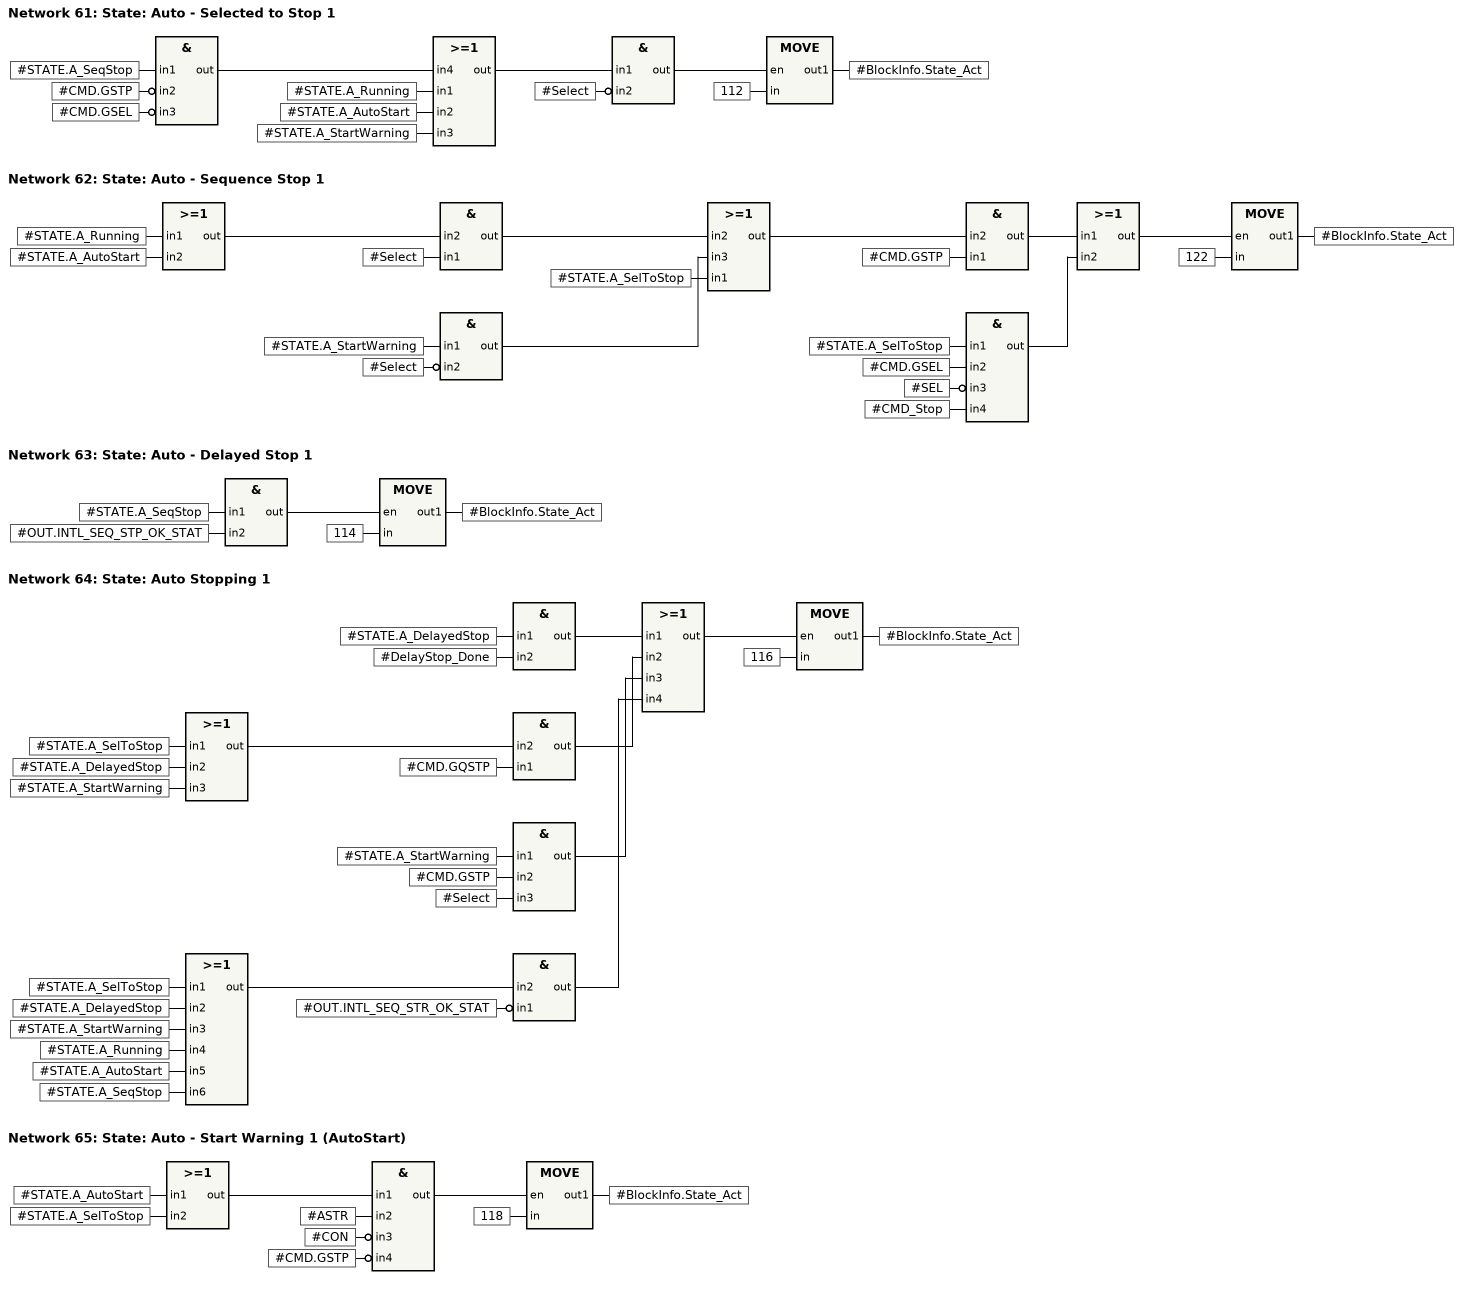
   IF ((#STATE.A_SeqStop AND NOT #CMD.GSTP AND NOT #CMD.GSEL) OR #STATE.A_Running OR #STATE.A_AutoStart OR #STATE.A_StartWarning) AND NOT #Select THEN
       #BlockInfo.State_Act := 112;
   END_IF;
END_REGION

REGION Network 62: State: Auto - Sequence Stop 1
   IF ((((#STATE.A_Running OR #STATE.A_AutoStart) AND #Select) OR (#STATE.A_StartWarning AND NOT #Select) OR #STATE.A_SelToStop) AND #CMD.GSTP) OR (#STATE.A_SelToStop AND #CMD.GSEL AND NOT #SEL AND #CMD_Stop) THEN
       #BlockInfo.State_Act := 122;
   END_IF;
END_REGION

REGION Network 63: State: Auto - Delayed Stop 1
   IF #STATE.A_SeqStop AND #OUT.INTL_SEQ_STP_OK_STAT THEN #BlockInfo.State_Act := 114; END_IF;
END_REGION

REGION Network 64: State: Auto Stopping 1
   IF (#STATE.A_DelayedStop AND #DelayStop_Done) OR ((#STATE.A_SelToStop OR #STATE.A_DelayedStop OR #STATE.A_StartWarning) AND #CMD.GQSTP) OR (#STATE.A_StartWarning AND #CMD.GSTP AND #Select) OR ((#STATE.A_SelToStop OR #STATE.A_DelayedStop OR #STATE.A_StartWarning OR #STATE.A_Running OR #STATE.A_AutoStart OR #STATE.A_SeqStop) AND NOT #OUT.INTL_SEQ_STR_OK_STAT) THEN
       #BlockInfo.State_Act := 116;
   END_IF;
END_REGION

REGION Network 65: State: Auto - Start Warning 1 (AutoStart)
   IF (#STATE.A_AutoStart OR #STATE.A_SelToStop) AND #ASTR AND NOT #CON AND NOT #CMD.GSTP THEN
       #BlockInfo.State_Act := 118;
   END_IF;
END_REGION

REGION Network 66
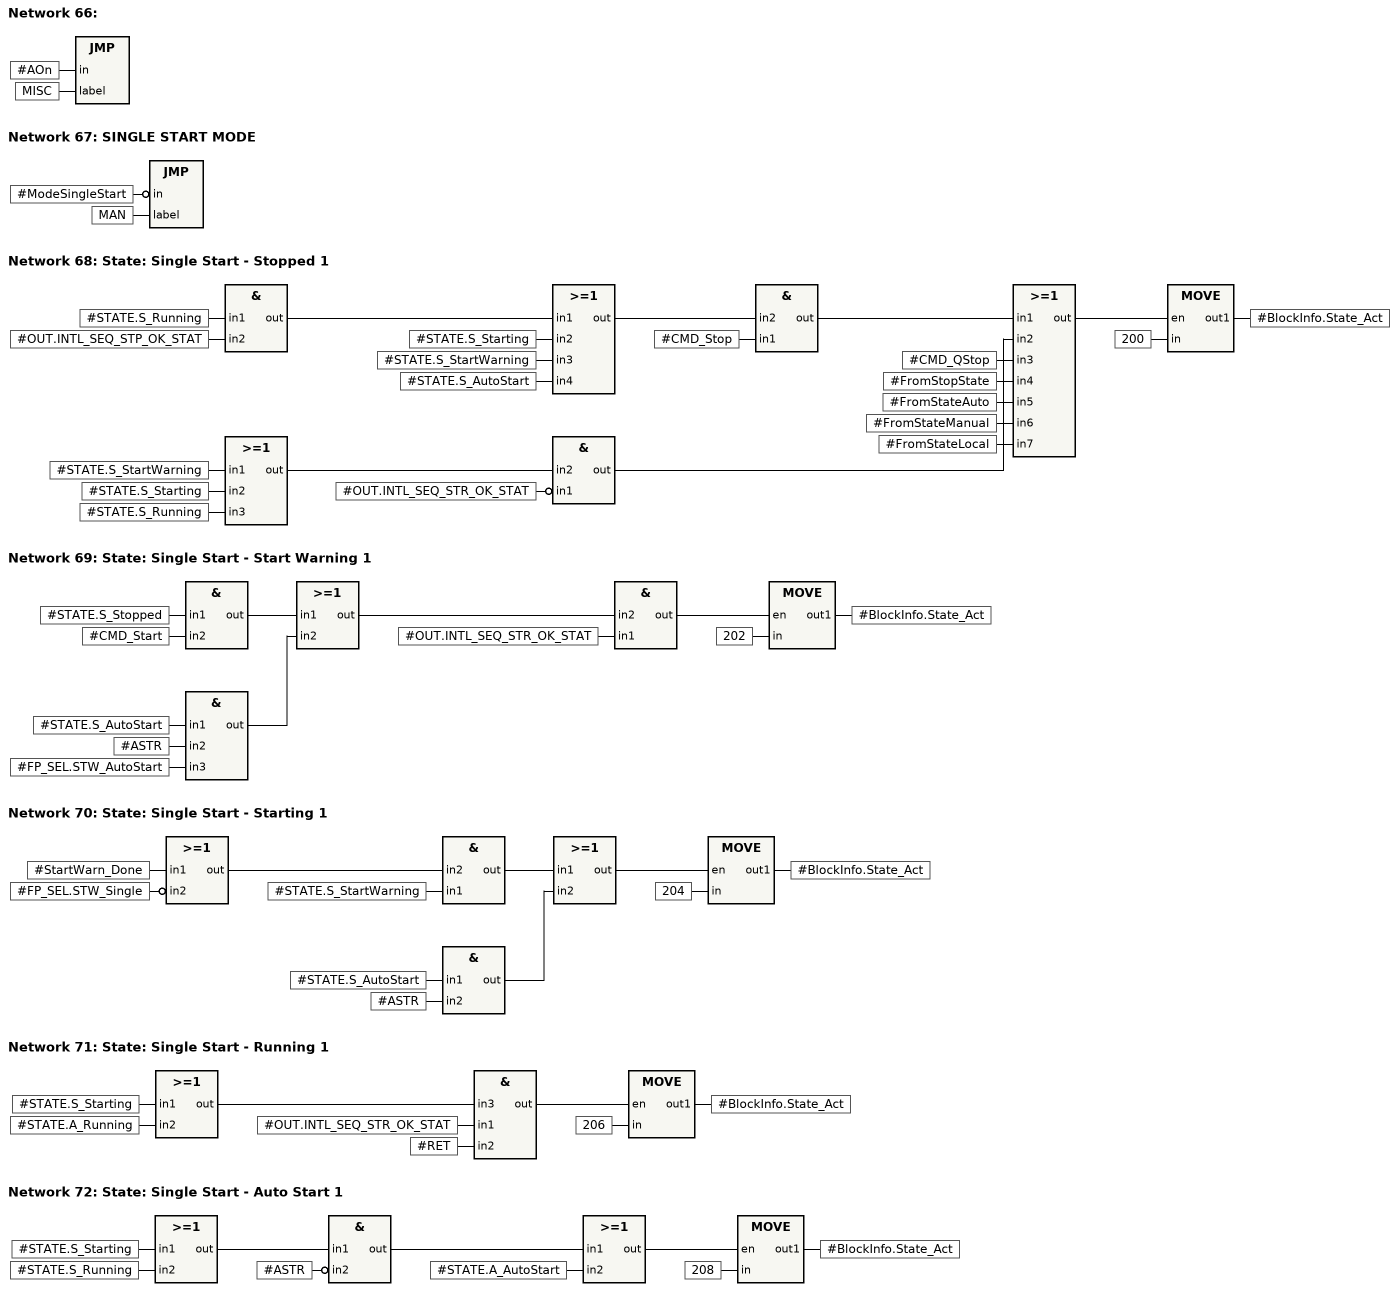
   IF #AOn THEN GOTO MISC; END_IF;
END_REGION

REGION Network 67: SINGLE START MODE
   SS1:
   IF NOT #ModeSingleStart THEN GOTO MAN; END_IF;
END_REGION

REGION Network 68: State: Single Start - Stopped 1
   IF (((#STATE.S_Running AND #OUT.INTL_SEQ_STP_OK_STAT) OR #STATE.S_Starting OR #STATE.S_StartWarning OR #STATE.S_AutoStart) AND #CMD_Stop) OR ((#STATE.S_StartWarning OR #STATE.S_Starting OR #STATE.S_Running) AND NOT #OUT.INTL_SEQ_STR_OK_STAT) OR #CMD_QStop OR #FromStopState OR #FromStateAuto OR #FromStateManual OR #FromStateLocal THEN
       #BlockInfo.State_Act := 200;
   END_IF;
END_REGION

REGION Network 69: State: Single Start - Start Warning 1
   IF ((#STATE.S_Stopped AND #CMD_Start) OR (#STATE.S_AutoStart AND #ASTR AND #FP_SEL.STW_AutoStart)) AND #OUT.INTL_SEQ_STR_OK_STAT THEN
       #BlockInfo.State_Act := 202;
   END_IF;
END_REGION

REGION Network 70: State: Single Start - Starting 1
   IF ((#StartWarn_Done OR NOT #FP_SEL.STW_Single) AND #STATE.S_StartWarning) OR (#STATE.S_AutoStart AND #ASTR) THEN
       #BlockInfo.State_Act := 204;
   END_IF;
END_REGION

REGION Network 71: State: Single Start - Running 1
   IF (#STATE.S_Starting OR #STATE.A_Running) AND #OUT.INTL_SEQ_STR_OK_STAT AND #RET THEN
       #BlockInfo.State_Act := 206;
   END_IF;
END_REGION

REGION Network 72: State: Single Start - Auto Start 1
   IF ((#STATE.S_Starting OR #STATE.S_Running) AND NOT #ASTR) OR #STATE.A_AutoStart THEN
       #BlockInfo.State_Act := 208;
   END_IF;
END_REGION

REGION Network 73
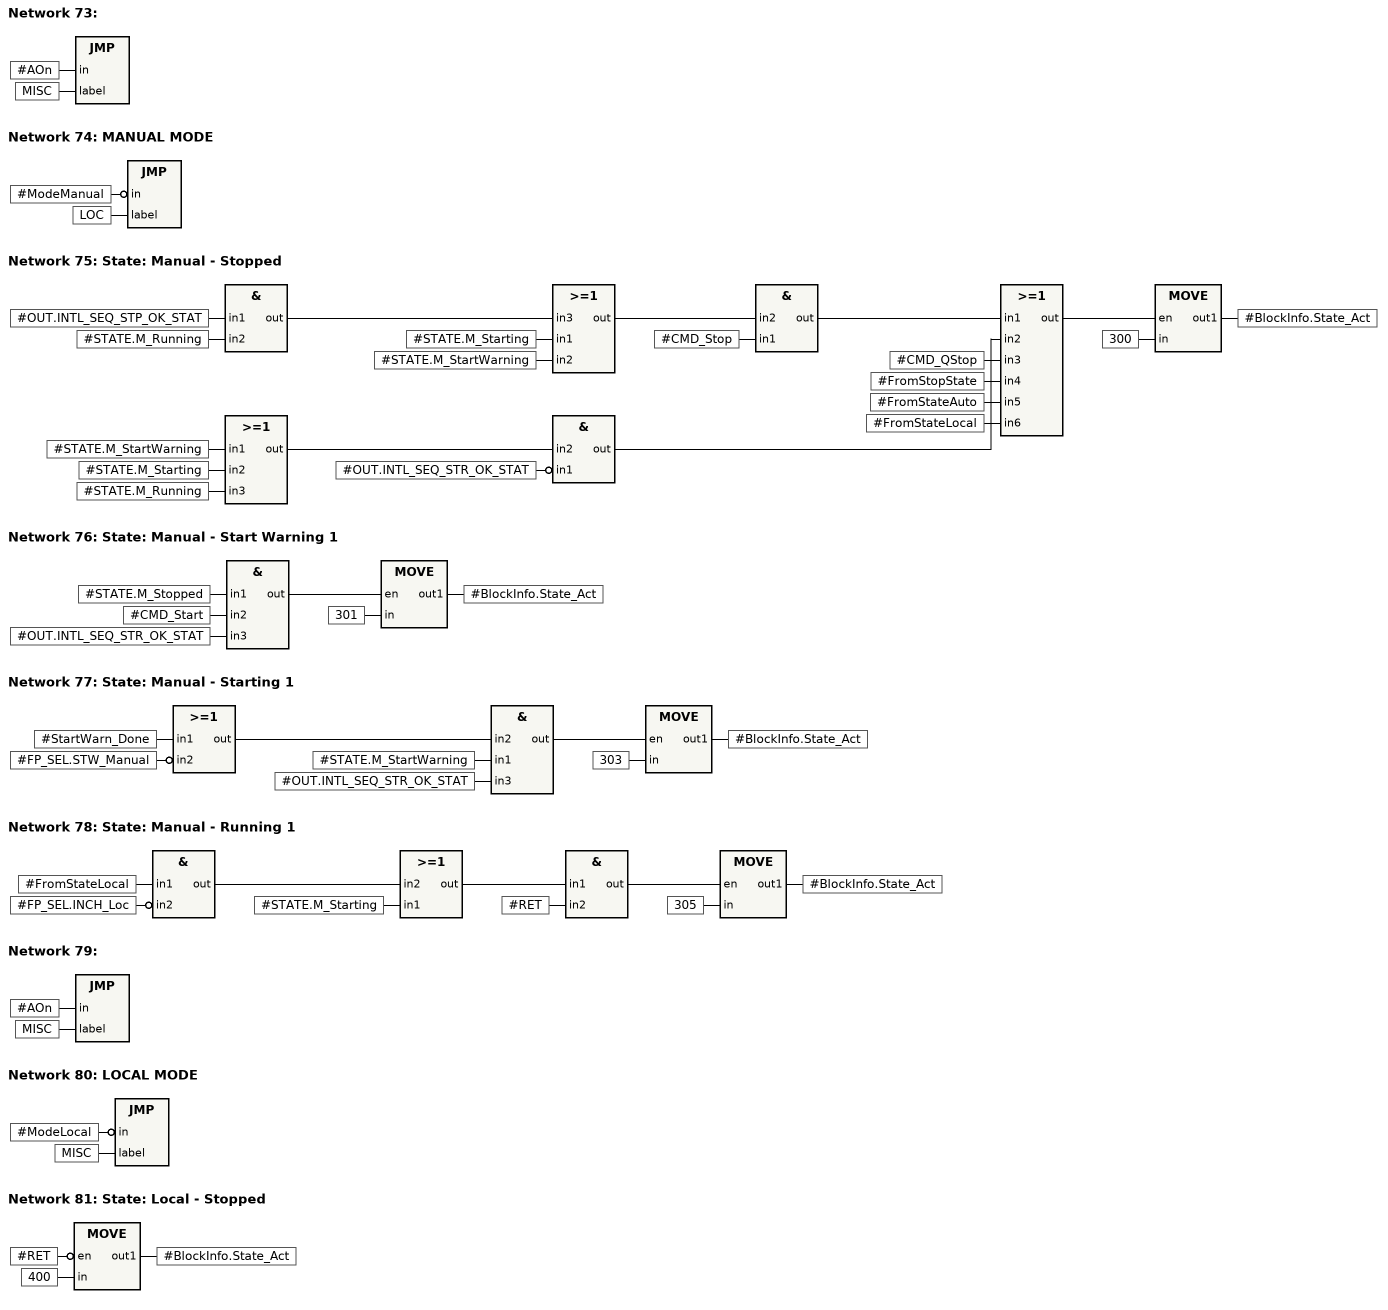
   IF #AOn THEN GOTO MISC; END_IF;
END_REGION

REGION Network 74: MANUAL MODE
   MAN:
   IF NOT #ModeManual THEN GOTO LOC; END_IF;
END_REGION

REGION Network 75: State: Manual - Stopped
   IF (((#OUT.INTL_SEQ_STP_OK_STAT AND #STATE.M_Running) OR #STATE.M_Starting OR #STATE.M_StartWarning) AND #CMD_Stop) OR ((#STATE.M_StartWarning OR #STATE.M_Starting OR #STATE.M_Running) AND NOT #OUT.INTL_SEQ_STR_OK_STAT) OR #CMD_QStop OR #FromStopState OR #FromStateAuto OR #FromStateLocal THEN
       #BlockInfo.State_Act := 300;
   END_IF;
END_REGION

REGION Network 76: State: Manual - Start Warning 1
   IF #STATE.M_Stopped AND #CMD_Start AND #OUT.INTL_SEQ_STR_OK_STAT THEN #BlockInfo.State_Act := 301; END_IF;
END_REGION

REGION Network 77: State: Manual - Starting 1
   IF (#StartWarn_Done OR NOT #FP_SEL.STW_Manual) AND #STATE.M_StartWarning AND #OUT.INTL_SEQ_STR_OK_STAT THEN
       #BlockInfo.State_Act := 303;
   END_IF;
END_REGION

REGION Network 78: State: Manual - Running 1
   IF ((#FromStateLocal AND NOT #FP_SEL.INCH_Loc) OR #STATE.M_Starting) AND #RET THEN
       #BlockInfo.State_Act := 305;
   END_IF;
END_REGION

REGION Network 79
   IF #AOn THEN GOTO MISC; END_IF;
END_REGION

REGION Network 80: LOCAL MODE
   LOC:
   IF NOT #ModeLocal THEN GOTO MISC; END_IF;
END_REGION

REGION Network 81: State: Local - Stopped
   IF NOT #RET THEN #BlockInfo.State_Act := 400; END_IF;
END_REGION

REGION Network 82: State: Local Running 1
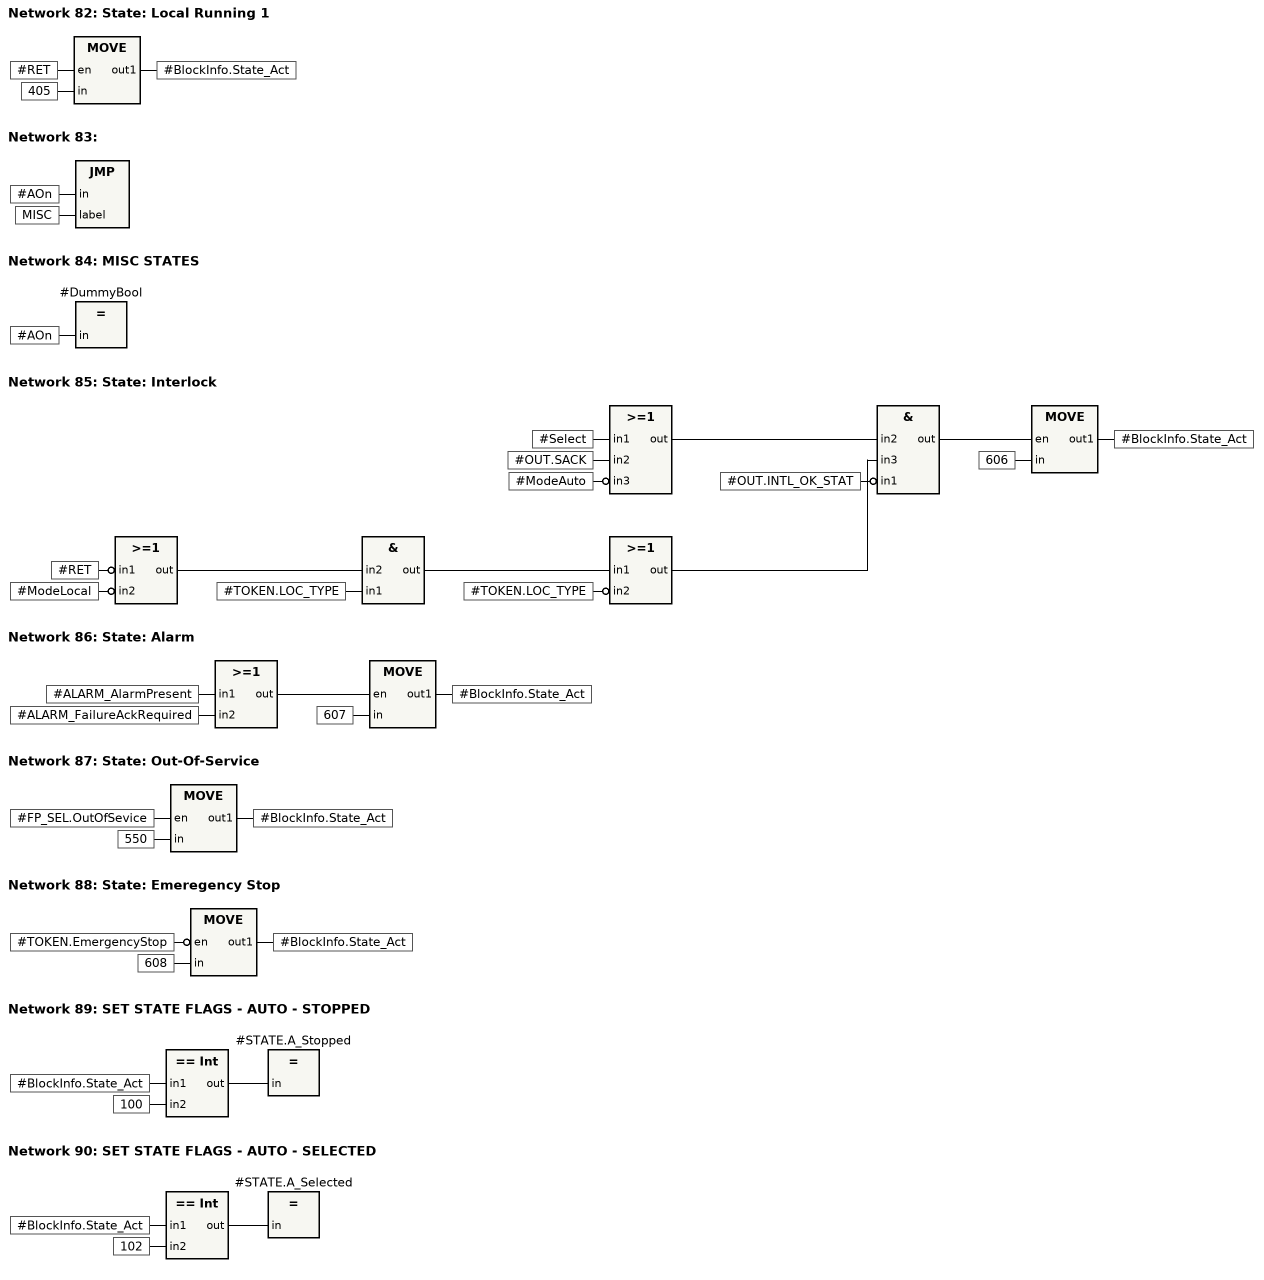
   IF #RET THEN #BlockInfo.State_Act := 405; END_IF;
END_REGION

REGION Network 83
   IF #AOn THEN GOTO MISC; END_IF;
END_REGION

REGION Network 84: MISC STATES
   MISC:
   #DummyBool := #AOn;
END_REGION

REGION Network 85: State: Interlock
   IF (#Select OR #OUT.SACK OR NOT #ModeAuto) AND (((NOT #RET OR NOT #ModeLocal) AND #TOKEN.LOC_TYPE) OR NOT #TOKEN.LOC_TYPE) AND NOT #OUT.INTL_OK_STAT THEN
       #BlockInfo.State_Act := 606;
   END_IF;
END_REGION

REGION Network 86: State: Alarm
   IF #ALARM_AlarmPresent OR #ALARM_FailureAckRequired THEN #BlockInfo.State_Act := 607; END_IF;
END_REGION

REGION Network 87: State: Out-Of-Service
   IF #FP_SEL.OutOfSevice THEN #BlockInfo.State_Act := 550; END_IF;
END_REGION

REGION Network 88: State: Emeregency Stop
   IF NOT #TOKEN.EmergencyStop THEN #BlockInfo.State_Act := 608; END_IF;
END_REGION

REGION Network 89: SET STATE FLAGS - AUTO - STOPPED
   #STATE.A_Stopped := #BlockInfo.State_Act = 100;
END_REGION

REGION Network 90: SET STATE FLAGS - AUTO - SELECTED
   #STATE.A_Selected := #BlockInfo.State_Act = 102;
END_REGION

REGION Network 91: SET STATE FLAGS - AUTO - SEQ START
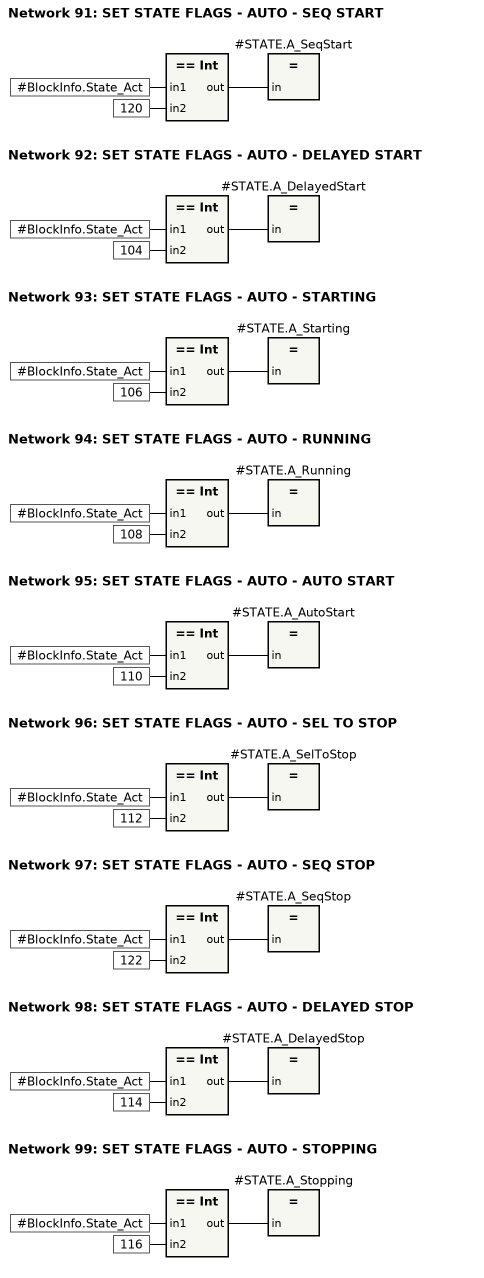
   #STATE.A_SeqStart := #BlockInfo.State_Act = 120;
END_REGION

REGION Network 92: SET STATE FLAGS - AUTO - DELAYED START
   #STATE.A_DelayedStart := #BlockInfo.State_Act = 104;
END_REGION

REGION Network 93: SET STATE FLAGS - AUTO - STARTING
   #STATE.A_Starting := #BlockInfo.State_Act = 106;
END_REGION

REGION Network 94: SET STATE FLAGS - AUTO - RUNNING
   #STATE.A_Running := #BlockInfo.State_Act = 108;
END_REGION

REGION Network 95: SET STATE FLAGS - AUTO - AUTO START
   #STATE.A_AutoStart := #BlockInfo.State_Act = 110;
END_REGION

REGION Network 96: SET STATE FLAGS - AUTO - SEL TO STOP
   #STATE.A_SelToStop := #BlockInfo.State_Act = 112;
END_REGION

REGION Network 97: SET STATE FLAGS - AUTO - SEQ STOP
   #STATE.A_SeqStop := #BlockInfo.State_Act = 122;
END_REGION

REGION Network 98: SET STATE FLAGS - AUTO - DELAYED STOP
   #STATE.A_DelayedStop := #BlockInfo.State_Act = 114;
END_REGION

REGION Network 99: SET STATE FLAGS - AUTO - STOPPING
   #STATE.A_Stopping := #BlockInfo.State_Act = 116;
END_REGION

REGION Network 100: SET STATE FLAGS - AUTO - START WARNING
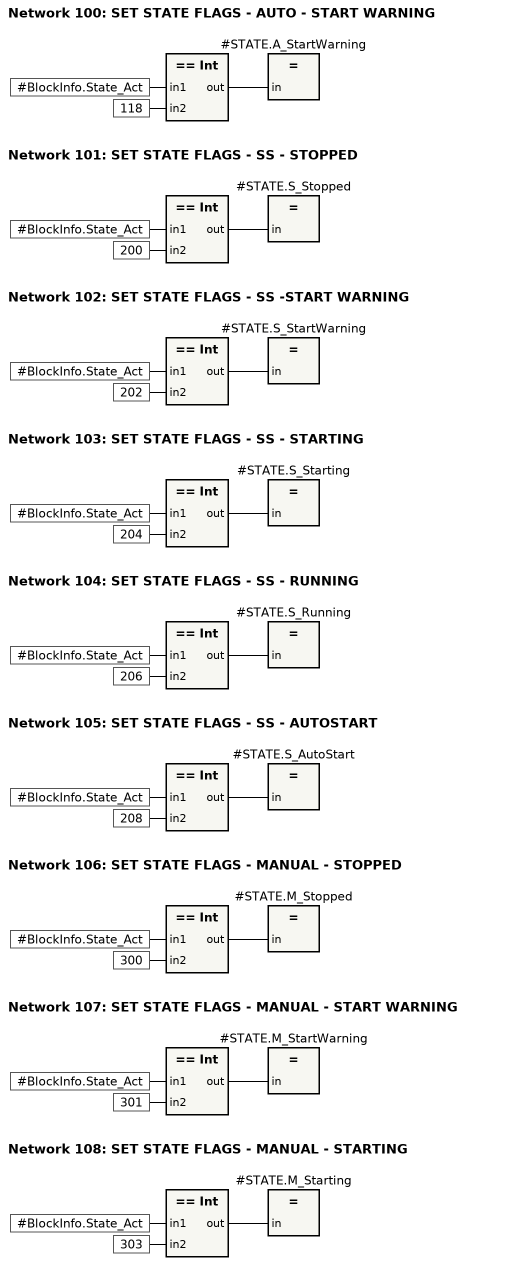
   #STATE.A_StartWarning := #BlockInfo.State_Act = 118;
END_REGION

REGION Network 101: SET STATE FLAGS - SS - STOPPED
   #STATE.S_Stopped := #BlockInfo.State_Act = 200;
END_REGION

REGION Network 102: SET STATE FLAGS - SS -START WARNING
   #STATE.S_StartWarning := #BlockInfo.State_Act = 202;
END_REGION

REGION Network 103: SET STATE FLAGS - SS - STARTING
   #STATE.S_Starting := #BlockInfo.State_Act = 204;
END_REGION

REGION Network 104: SET STATE FLAGS - SS - RUNNING
   #STATE.S_Running := #BlockInfo.State_Act = 206;
END_REGION

REGION Network 105: SET STATE FLAGS - SS - AUTOSTART
   #STATE.S_AutoStart := #BlockInfo.State_Act = 208;
END_REGION

REGION Network 106: SET STATE FLAGS - MANUAL - STOPPED
   #STATE.M_Stopped := #BlockInfo.State_Act = 300;
END_REGION

REGION Network 107: SET STATE FLAGS - MANUAL - START WARNING
   #STATE.M_StartWarning := #BlockInfo.State_Act = 301;
END_REGION

REGION Network 108: SET STATE FLAGS - MANUAL - STARTING
   #STATE.M_Starting := #BlockInfo.State_Act = 303;
END_REGION

REGION Network 109: SET STATE FLAGS - MANUAL - RUNNING
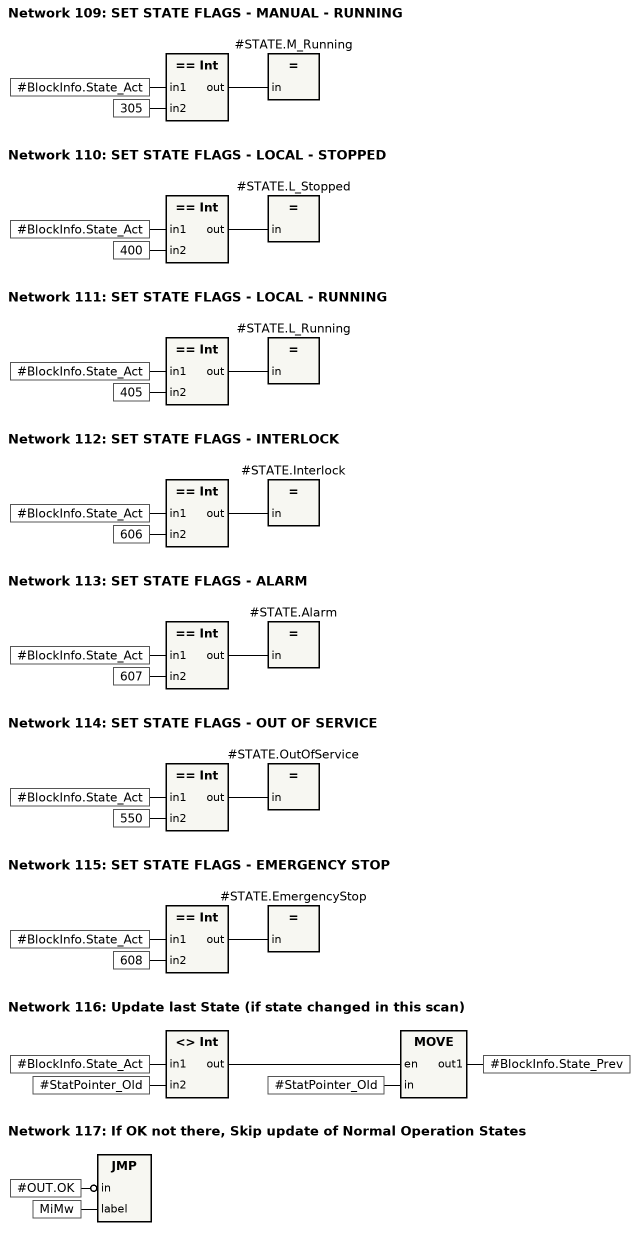
   #STATE.M_Running := #BlockInfo.State_Act = 305;
END_REGION

REGION Network 110: SET STATE FLAGS - LOCAL - STOPPED
   #STATE.L_Stopped := #BlockInfo.State_Act = 400;
END_REGION

REGION Network 111: SET STATE FLAGS - LOCAL - RUNNING
   #STATE.L_Running := #BlockInfo.State_Act = 405;
END_REGION

REGION Network 112: SET STATE FLAGS - INTERLOCK
   #STATE.Interlock := #BlockInfo.State_Act = 606;
END_REGION

REGION Network 113: SET STATE FLAGS - ALARM
   #STATE.Alarm := #BlockInfo.State_Act = 607;
END_REGION

REGION Network 114: SET STATE FLAGS - OUT OF SERVICE
   #STATE.OutOfService := #BlockInfo.State_Act = 550;
END_REGION

REGION Network 115: SET STATE FLAGS - EMERGENCY STOP
   #STATE.EmergencyStop := #BlockInfo.State_Act = 608;
END_REGION

REGION Network 116: Update last State (if state changed in this scan)
   IF #BlockInfo.State_Act <> #StatPointer_Old THEN #BlockInfo.State_Prev := #StatPointer_Old; END_IF;
END_REGION

REGION Network 117: If OK not there, Skip update of Normal Operation States
   // Build 006 - 30.09.2020 (EXTBOB): Skipped Normal MSW status update in case of Alarm Condition, Newly Added
   IF NOT #OUT.OK THEN GOTO MiMw; END_IF;
END_REGION

REGION Network 118: UPDATE MSW
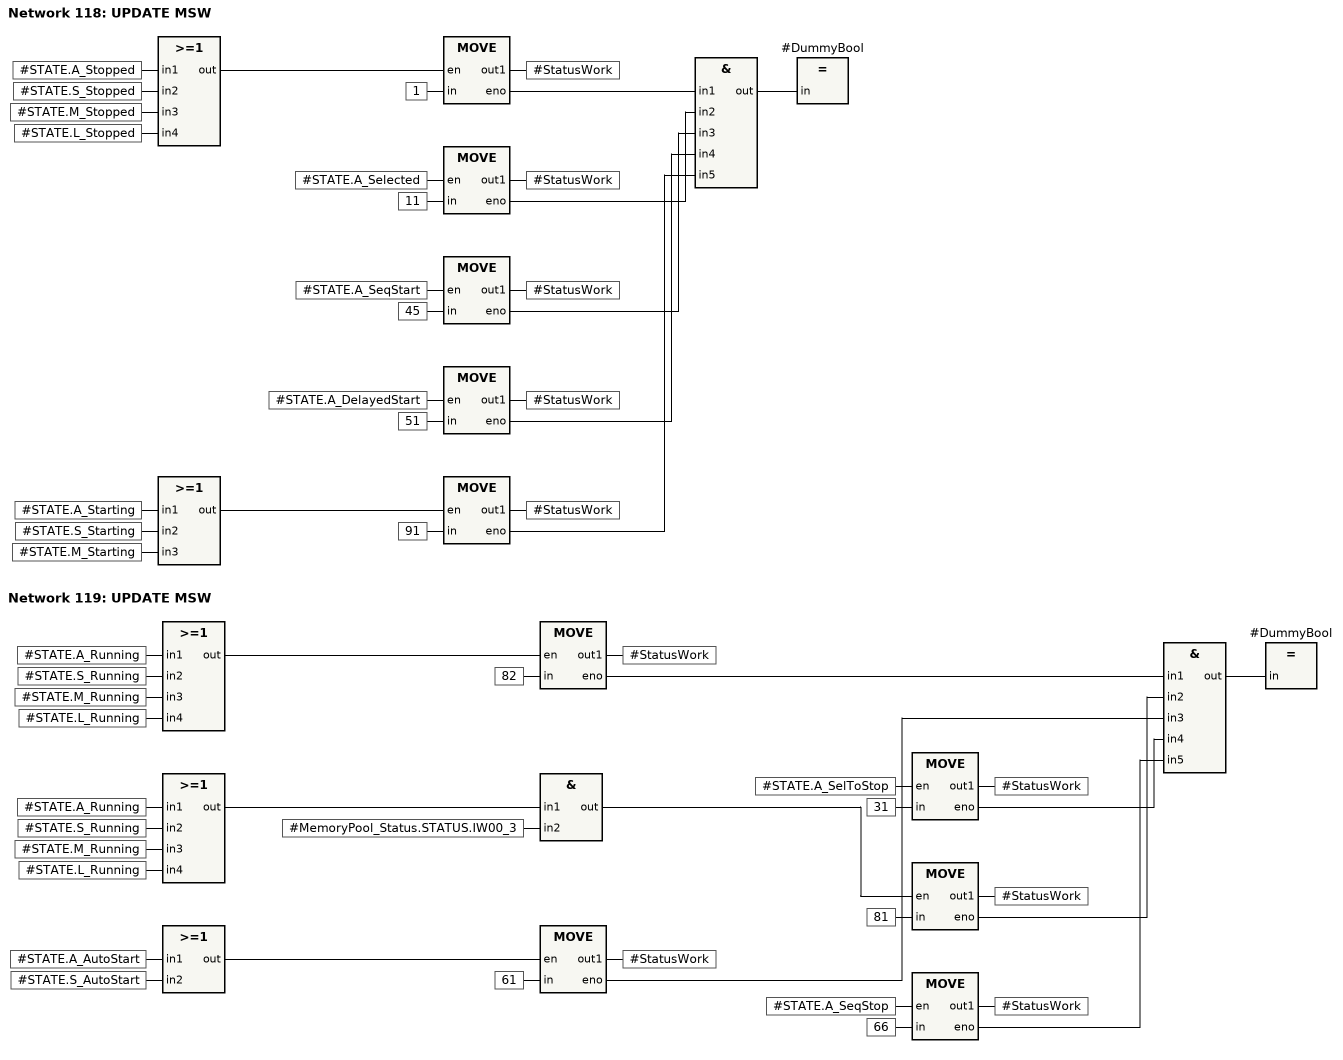
   // ENO of a box is taken as its EN; it also drops when the box reports an error
   #_w1 := #STATE.A_Stopped OR #STATE.S_Stopped OR #STATE.M_Stopped OR #STATE.L_Stopped;
   IF #_w1 THEN #StatusWork := 1; END_IF;
   IF #STATE.A_Selected THEN #StatusWork := 11; END_IF;
   IF #STATE.A_SeqStart THEN #StatusWork := 45; END_IF;
   IF #STATE.A_DelayedStart THEN #StatusWork := 51; END_IF;
   #_w2 := #STATE.A_Starting OR #STATE.S_Starting OR #STATE.M_Starting;
   IF #_w2 THEN #StatusWork := 91; END_IF;
   #DummyBool := #_w1 AND #STATE.A_Selected AND #STATE.A_SeqStart AND #STATE.A_DelayedStart AND #_w2;
END_REGION

REGION Network 119: UPDATE MSW
   // ENO of a box is taken as its EN; it also drops when the box reports an error
   #_w1 := #STATE.A_Running OR #STATE.S_Running OR #STATE.M_Running OR #STATE.L_Running;
   IF #_w1 THEN #StatusWork := 82; END_IF;
   #_w2 := (#STATE.A_Running OR #STATE.S_Running OR #STATE.M_Running OR #STATE.L_Running) AND #MemoryPool_Status.STATUS.IW00_3;
   IF #_w2 THEN #StatusWork := 81; END_IF;
   #_w3 := #STATE.A_AutoStart OR #STATE.S_AutoStart;
   IF #_w3 THEN #StatusWork := 61; END_IF;
   IF #STATE.A_SelToStop THEN #StatusWork := 31; END_IF;
   IF #STATE.A_SeqStop THEN #StatusWork := 66; END_IF;
   #DummyBool := #_w1 AND #_w2 AND #_w3 AND #STATE.A_SelToStop AND #STATE.A_SeqStop;
END_REGION

REGION Network 120
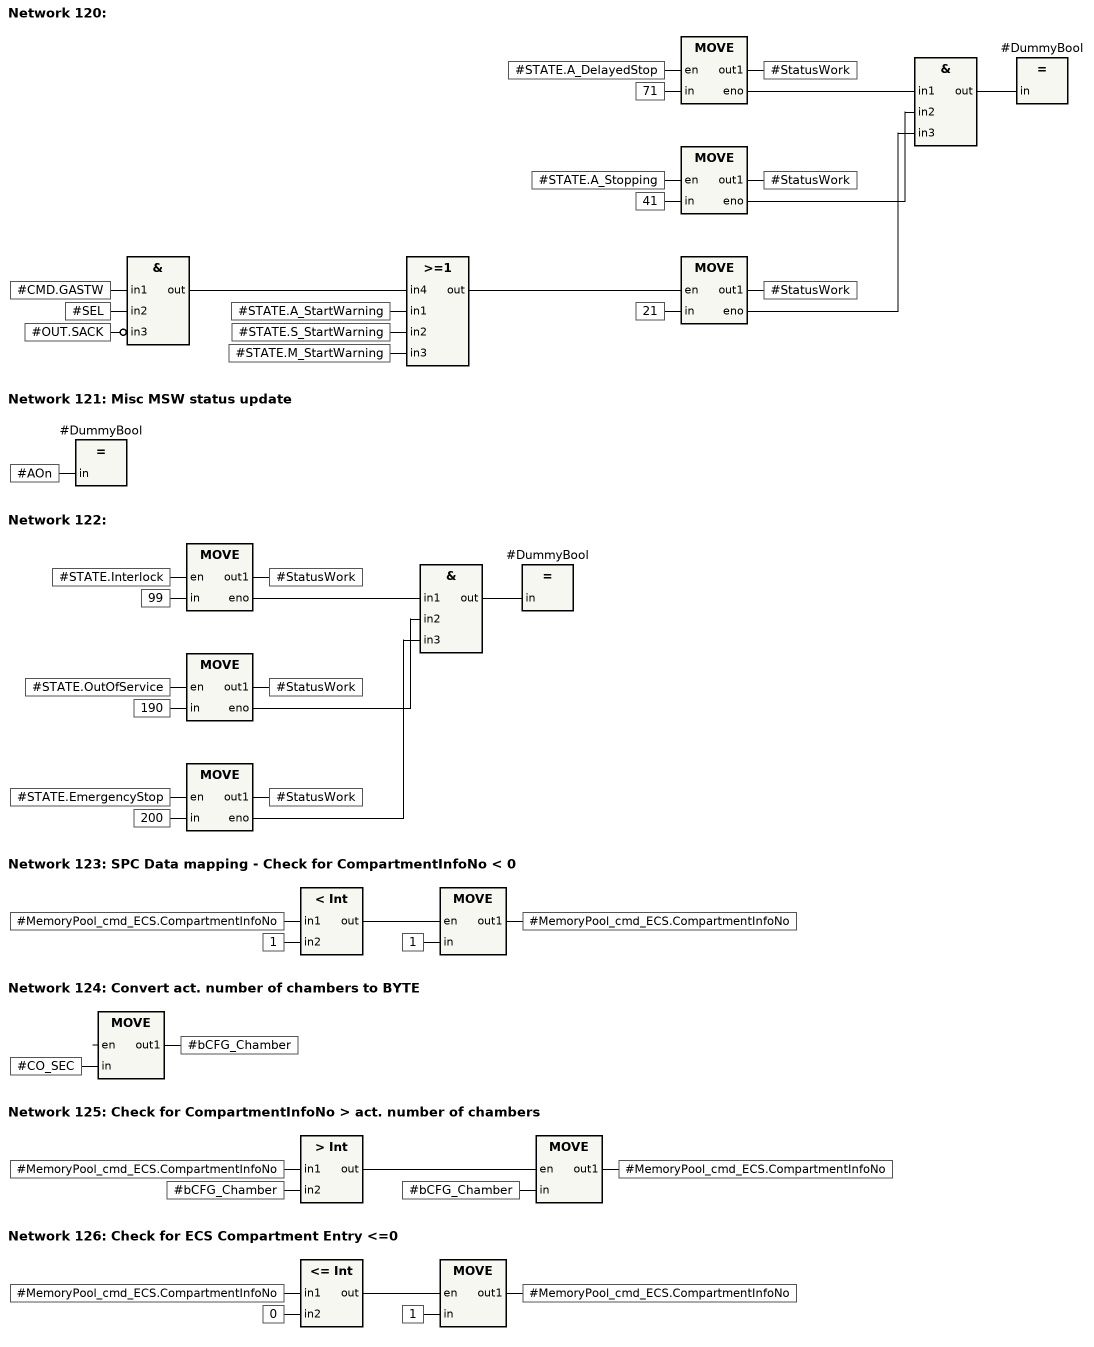
   // ENO of a box is taken as its EN; it also drops when the box reports an error
   IF #STATE.A_DelayedStop THEN #StatusWork := 71; END_IF;
   IF #STATE.A_Stopping THEN #StatusWork := 41; END_IF;
   #_w1 := (#CMD.GASTW AND #SEL AND NOT #OUT.SACK) OR #STATE.A_StartWarning OR #STATE.S_StartWarning OR #STATE.M_StartWarning;
   IF #_w1 THEN #StatusWork := 21; END_IF;
   #DummyBool := #STATE.A_DelayedStop AND #STATE.A_Stopping AND #_w1;
END_REGION

REGION Network 121: Misc MSW status update
   // Build 006 - 30.09.2020 (EXTBOB): Skipped Normal MSW status update in case of Alarm Condition, Newly Added
   MiMw:
   #DummyBool := #AOn;
END_REGION

REGION Network 122
   // ENO of a box is taken as its EN; it also drops when the box reports an error
   IF #STATE.Interlock THEN #StatusWork := 99; END_IF;
   IF #STATE.OutOfService THEN #StatusWork := 190; END_IF;
   IF #STATE.EmergencyStop THEN #StatusWork := 200; END_IF;
   #DummyBool := #STATE.Interlock AND #STATE.OutOfService AND #STATE.EmergencyStop;
END_REGION

REGION Network 123: SPC Data mapping - Check for CompartmentInfoNo < 0
   IF #MemoryPool_cmd_ECS.CompartmentInfoNo < 1 THEN #MemoryPool_cmd_ECS.CompartmentInfoNo := 1; END_IF;
END_REGION

REGION Network 124: Convert act. number of chambers to BYTE
   #bCFG_Chamber := #CO_SEC;
END_REGION

REGION Network 125: Check for CompartmentInfoNo > act. number of chambers
   IF #MemoryPool_cmd_ECS.CompartmentInfoNo > #bCFG_Chamber THEN
       #MemoryPool_cmd_ECS.CompartmentInfoNo := #bCFG_Chamber;
   END_IF;
END_REGION

REGION Network 126: Check for ECS Compartment Entry <=0
   IF #MemoryPool_cmd_ECS.CompartmentInfoNo <= 0 THEN #MemoryPool_cmd_ECS.CompartmentInfoNo := 1; END_IF;
END_REGION

REGION Network 127: Convert IO_Addr from INT to WORD
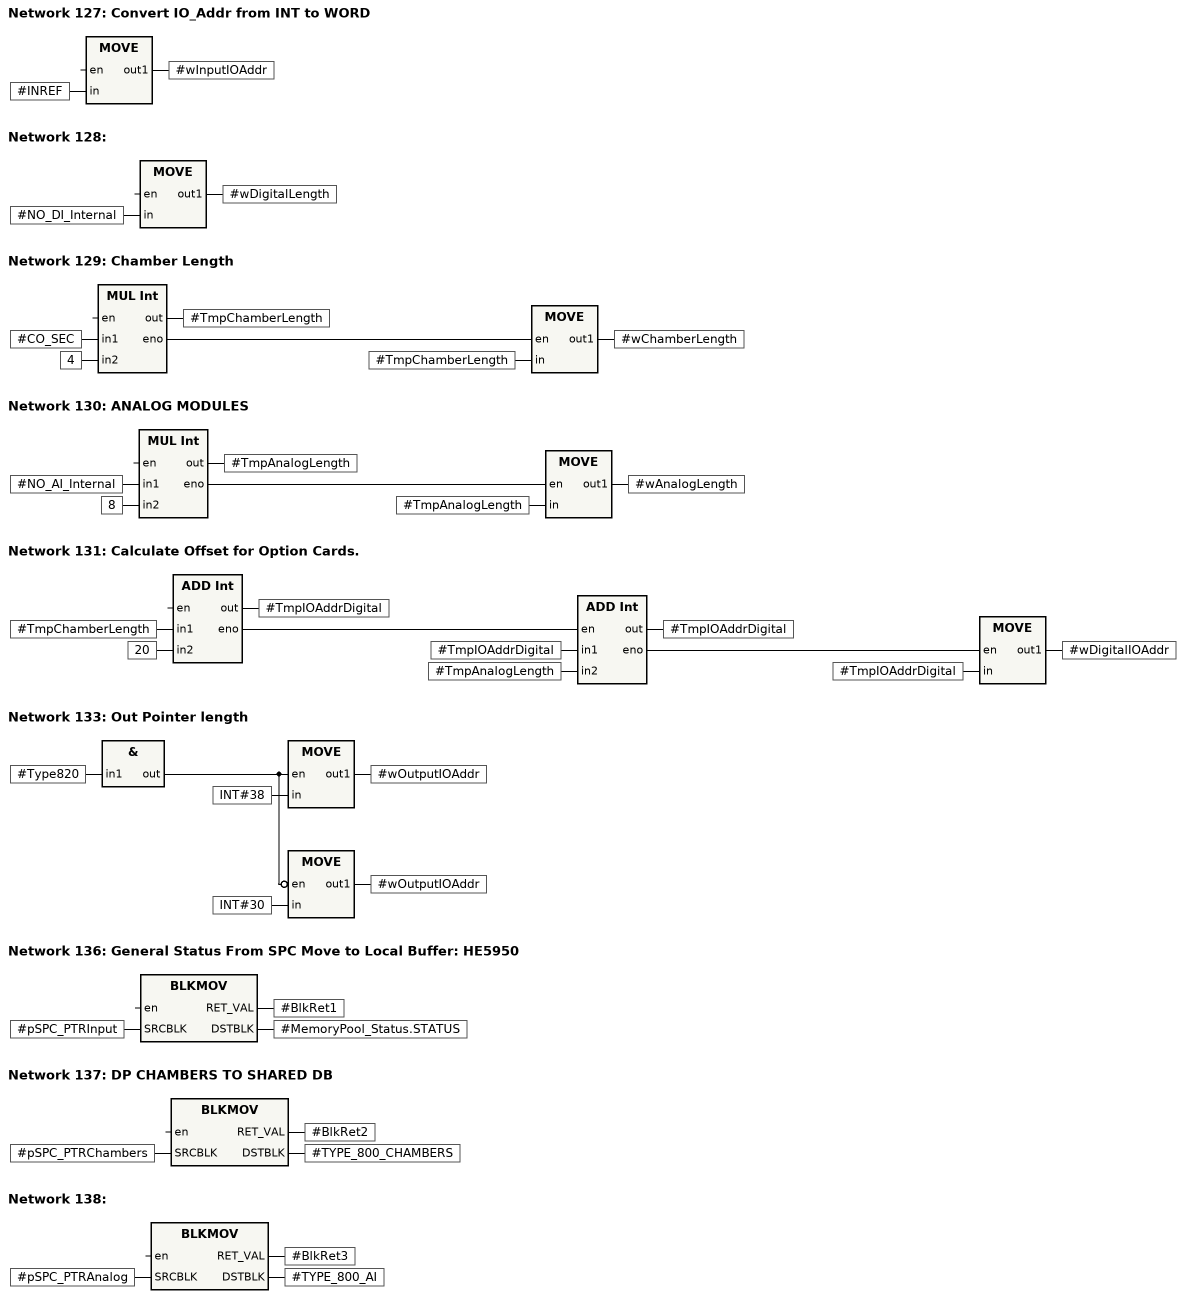
   #wInputIOAddr := #INREF;
END_REGION

REGION Network 128
   // Build 007 - 03.12.2020 (VIV-IN): NO_AI_Internal changed to NO_DI_Internal typo 
   // error corrected
   #wDigitalLength := #NO_DI_Internal;
END_REGION

REGION Network 129: Chamber Length
   // Calculate amount of bytes for the number of chambers
   // ENO of a box is taken as its EN; it also drops when the box reports an error
   #TmpChamberLength := #CO_SEC * 4;
   #wChamberLength := #TmpChamberLength;
END_REGION

REGION Network 130: ANALOG MODULES
   // Length In Bytes
   // ENO of a box is taken as its EN; it also drops when the box reports an error
   #TmpAnalogLength := #NO_AI_Internal * 8;
   #wAnalogLength := #TmpAnalogLength;
END_REGION

REGION Network 131: Calculate Offset for Option Cards.
   // Temp05MulVal is the length of chamber data. DIGITAL Option Card lies after 
   // chamber data and AI card.
   // ENO of a box is taken as its EN; it also drops when the box reports an error
   #TmpIOAddrDigital := #TmpChamberLength + 20;
   #TmpIOAddrDigital := #TmpIOAddrDigital + #TmpAnalogLength;
   #wDigitalIOAddr := #TmpIOAddrDigital;
END_REGION

REGION Network 132 (STL): POINTER CONSTRUCTION
   // Pointer for Bag Filter Controller Input Image 0-19 BYTE OFFSET
         LAR1;

         L     16#10;  //Syntax ID
         T     LB[AR1, P#0.0];

         L     16#02;  // Data Type= BYTE
         T     LB[AR1, P#1.0];

         L     20;
         T     LW[AR1, P#2.0];  //0..19 DATA BYTES TO TRANSFER

         L     0;
         T     LW[AR1, P#4.0];  //Not Used

         L     #INREF;  // Source offset (Variable for Node's)
         SLD   3;  // with offset
         OD    16#8100_0000;  // Input Area (I/O) Code (S7)
         T     LD[AR1, P#6.0];  // ..Store byte 6/7/8/9
         NOP   0;

         LAR1;

         L     16#10;  //Syntax ID
         T     LB[AR1, P#0.0];

         L     16#02;  // Data Type= BYTE
         T     LB[AR1, P#1.0];

         L     #wChamberLength;
         T     LW[AR1, P#2.0];  //0..Chamber length DATA BYTES TO TRANSFER

         L     0;
         T     LW[AR1, P#4.0];  //Not Used

         L     #INREF;  // Source offset (Variable for Node's)
         L     20;  //System offset
         +I;
         SLD   3;  // with offset
         OD    16#8100_0000;  // Input Area (I/O) Code (S7)
         T     LD[AR1, P#6.0];  // ..Store byte 6/7/8/9
         NOP   0;

   //Analog IO Address
         LAR1;

         L     16#10;  //Syntax ID
         T     LB[AR1, P#0.0];

         L     16#02;  // Data Type= bytes
         T     LB[AR1, P#1.0];

         L     #wAnalogLength;
         T     LW[AR1, P#2.0];  //0..Analog lenght DATA BYTES TO TRANSFER

         L     0;
         T     LW[AR1, P#4.0];  //Not Used

         L     #INREF;  // Source offset (Variable for Node's)
         L     #wChamberLength;
         +I;
         L     20;  //System offset
         +I;
         SLD   3;  // with offset
         OD    16#8100_0000;  // Input Area (I/O) Code (S7)
         T     LD[AR1, P#6.0];  // ..Store byte 6/7/8/9
         NOP   0;
END_REGION

REGION Network 133: Out Pointer length
   // - SPC820 -> 38 Bytes, Other Controller - 30 bytes
   IF #Type820 THEN #wOutputIOAddr := INT#38; END_IF;
   IF NOT #Type820 THEN #wOutputIOAddr := INT#30; END_IF;
END_REGION

REGION Network 134 (STL): POINTER CONSTRUCTION
   // Pointer for Bag Filter Controller Output Image 0-29 BYTE OFFSET
         LAR1;

         L     16#10;  //Syntax ID
         T     LB[AR1, P#0.0];

         L     16#02;  // Data Type= BYTE
         T     LB[AR1, P#1.0];

         L     #wOutputIOAddr;
         T     LW[AR1, P#2.0];  //0..29 DATA BYTES TO TRANSFER

         L     0;
         T     LW[AR1, P#4.0];  //Not Used For Memory Area

         L     #OUTREF;  // Source offset (Variable for Node's)
         SLD   3;  // with offset
         OD    16#8200_0000;  // Input Area (I/O) Code (S7)
         T     LD[AR1, P#6.0];  // ..Store byte 6/7/8/9
         NOP   0;
END_REGION

REGION Network 135 (STL): POINTER CONSTRUCTION
   // Pointer for Digital Cards in the SPC
         LAR1;

         L     16#10;  //Syntax ID
         T     LB[AR1, P#0.0];

         L     16#02;  // Data Type= bytes
         T     LB[AR1, P#1.0];

         L     #wDigitalLength;
         T     LW[AR1, P#2.0];  //1 DATA BYTES/CARD TO TRANSFER

         L     0;
         T     LW[AR1, P#4.0];  //Not Used

         L     #INREF;  // Source offset (Variable for Node's)
         L     #wDigitalIOAddr;  // Source offset (Variable for Node's)
         +I;
         SLD   3;  // with offset
         OD    16#8100_0000;  // Input Area (I/O) Code (S7)
         T     LD[AR1, P#6.0];  // ..Store byte 6/7/8/9
         NOP   0;
END_REGION

REGION Network 136: General Status From SPC Move to Local Buffer: HE5950
   #BlkRet1 := BLKMOV(SRCBLK := #pSPC_PTRInput, DSTBLK => #MemoryPool_Status.STATUS);
END_REGION

REGION Network 137: DP CHAMBERS TO SHARED DB
   // Mvespc chamber data Local data
   // If Filter is Model 800 then Run This Block Call
   #BlkRet2 := BLKMOV(SRCBLK := #pSPC_PTRChambers, DSTBLK => #TYPE_800_CHAMBERS);
END_REGION

REGION Network 138
   // Move Analog Data to Local data
   #BlkRet3 := BLKMOV(SRCBLK := #pSPC_PTRAnalog, DSTBLK => #TYPE_800_AI);
END_REGION

REGION Network 139: DP DIGITAL TO SHARED DB
   // Move digital card data to Local data
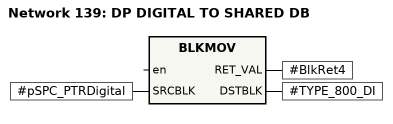
   #BlkRet4 := BLKMOV(SRCBLK := #pSPC_PTRDigital, DSTBLK => #TYPE_800_DI);
END_REGION

REGION Network 140: Convert Analog to Floating Point
   // Transfer all Word data into Double Format and then to Real. Multiply with 10.0
   // SPC must be configured for sending processvalue with floating point 
   // representation.
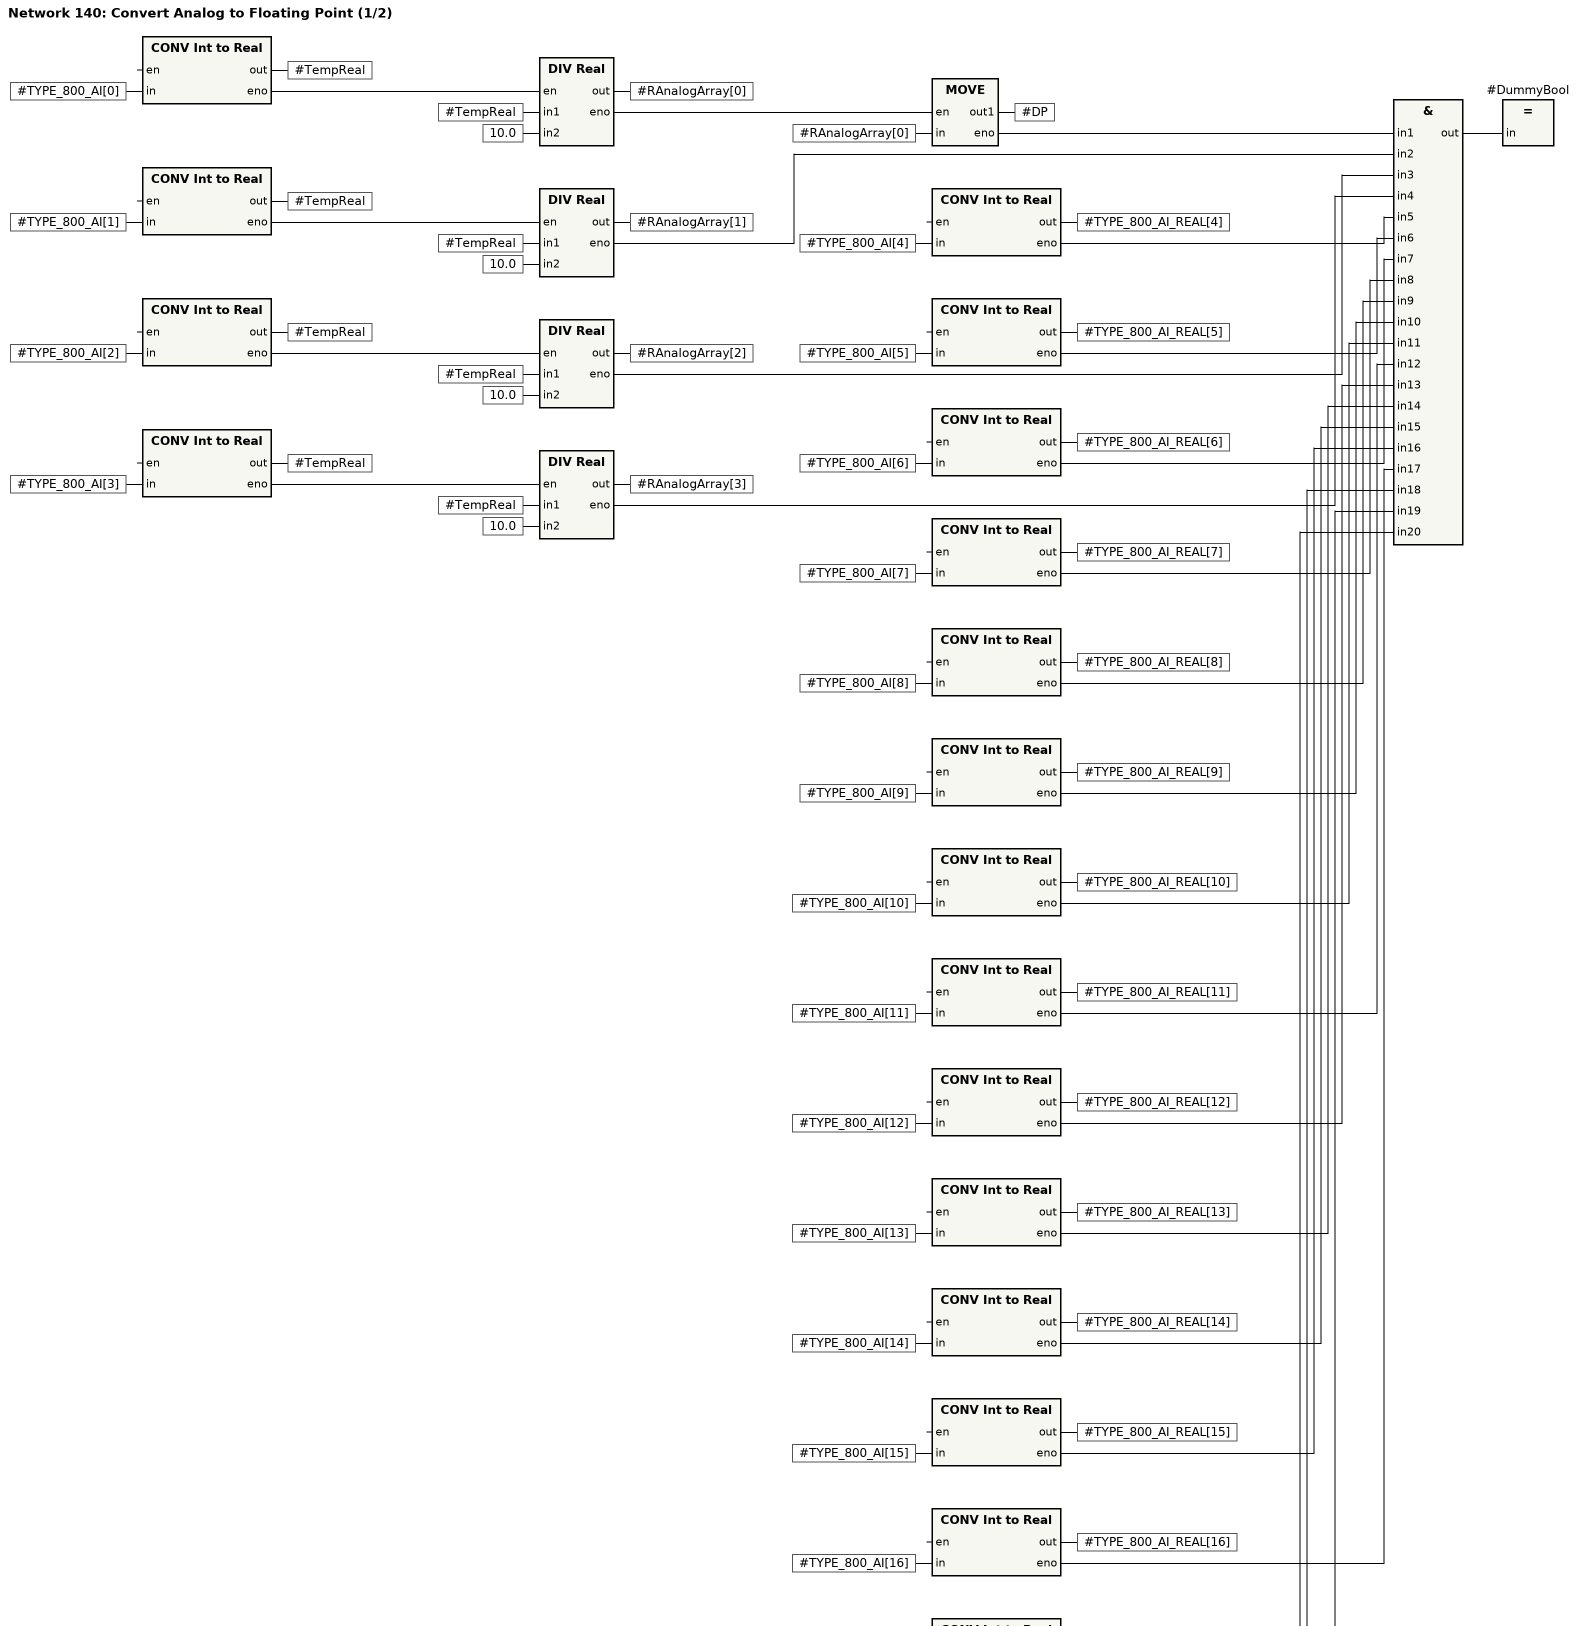
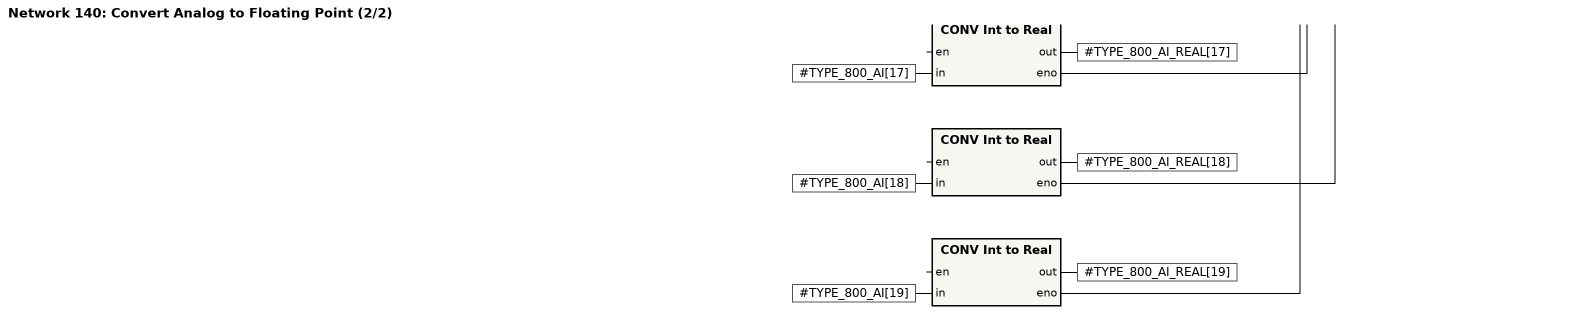
   #TempReal := INT_TO_REAL(#TYPE_800_AI[0]);
   #RAnalogArray[0] := #TempReal / 10.0;
   #DP := #RAnalogArray[0];
   #TempReal := INT_TO_REAL(#TYPE_800_AI[1]);
   #RAnalogArray[1] := #TempReal / 10.0;
   #TempReal := INT_TO_REAL(#TYPE_800_AI[2]);
   #RAnalogArray[2] := #TempReal / 10.0;
   #TempReal := INT_TO_REAL(#TYPE_800_AI[3]);
   #RAnalogArray[3] := #TempReal / 10.0;
   #TYPE_800_AI_REAL[4] := INT_TO_REAL(#TYPE_800_AI[4]);
   #TYPE_800_AI_REAL[5] := INT_TO_REAL(#TYPE_800_AI[5]);
   #TYPE_800_AI_REAL[6] := INT_TO_REAL(#TYPE_800_AI[6]);
   #TYPE_800_AI_REAL[7] := INT_TO_REAL(#TYPE_800_AI[7]);
   #TYPE_800_AI_REAL[8] := INT_TO_REAL(#TYPE_800_AI[8]);
   #TYPE_800_AI_REAL[9] := INT_TO_REAL(#TYPE_800_AI[9]);
   #TYPE_800_AI_REAL[10] := INT_TO_REAL(#TYPE_800_AI[10]);
   #TYPE_800_AI_REAL[11] := INT_TO_REAL(#TYPE_800_AI[11]);
   #TYPE_800_AI_REAL[12] := INT_TO_REAL(#TYPE_800_AI[12]);
   #TYPE_800_AI_REAL[13] := INT_TO_REAL(#TYPE_800_AI[13]);
   #TYPE_800_AI_REAL[14] := INT_TO_REAL(#TYPE_800_AI[14]);
   #TYPE_800_AI_REAL[15] := INT_TO_REAL(#TYPE_800_AI[15]);
   #TYPE_800_AI_REAL[16] := INT_TO_REAL(#TYPE_800_AI[16]);
   #TYPE_800_AI_REAL[17] := INT_TO_REAL(#TYPE_800_AI[17]);
   #TYPE_800_AI_REAL[18] := INT_TO_REAL(#TYPE_800_AI[18]);
   #TYPE_800_AI_REAL[19] := INT_TO_REAL(#TYPE_800_AI[19]);
   #DummyBool := TRUE;
END_REGION

REGION Network 141
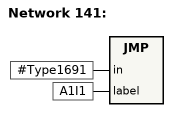
   IF #Type1691 THEN GOTO A1I1; END_IF;
END_REGION

REGION Network 142: Convert Analog to Floating Point
   // Transfer all Word data into Double Format and then to Real. Multiply with 10.0
   // SPC must be configured for sending processvalue with floating point 
   // representation
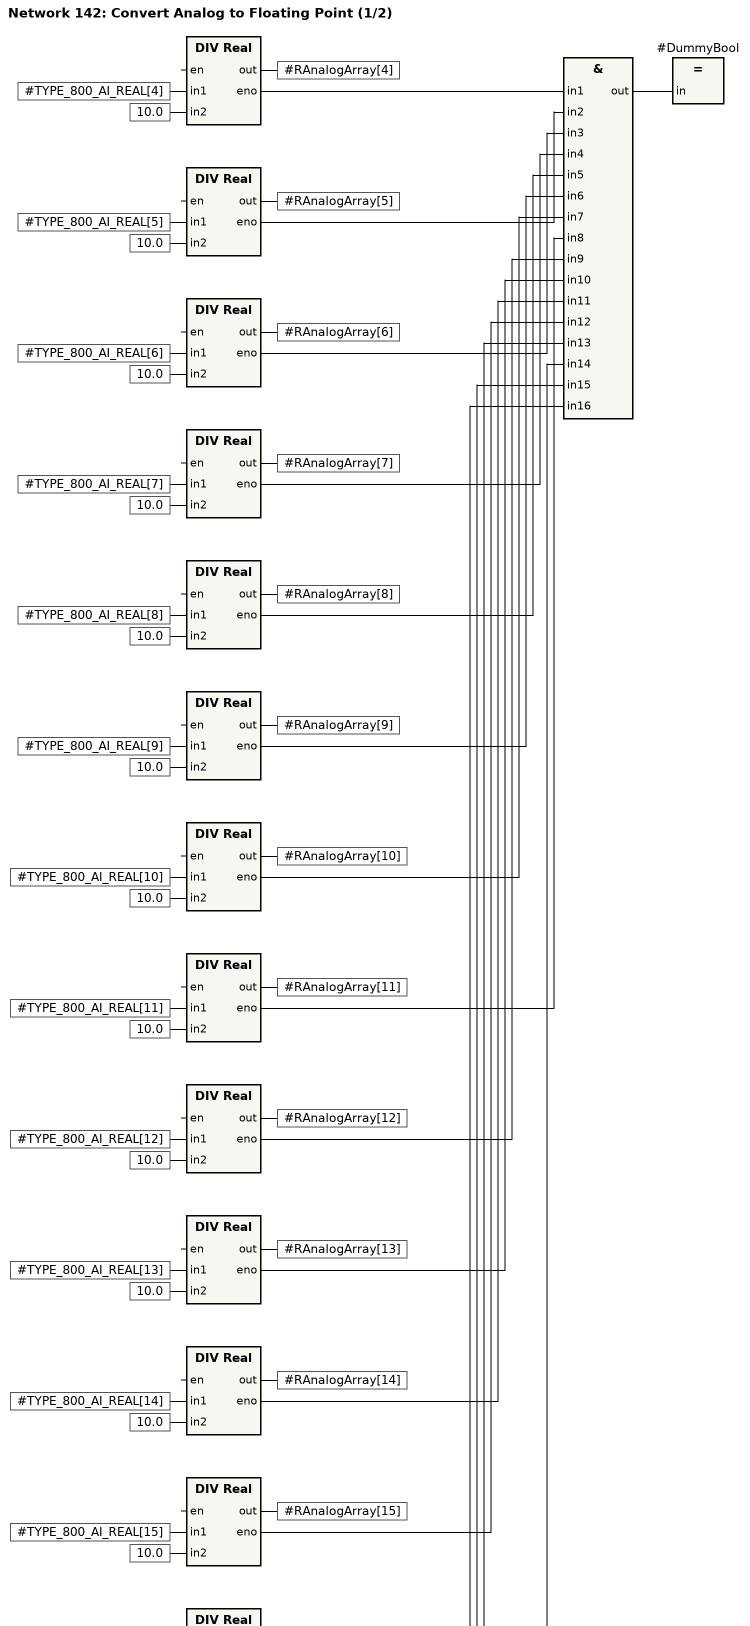
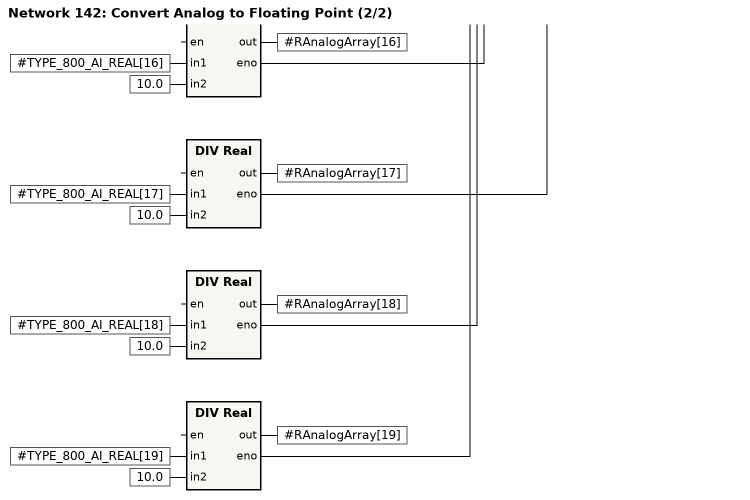
   #RAnalogArray[4] := #TYPE_800_AI_REAL[4] / 10.0;
   #RAnalogArray[5] := #TYPE_800_AI_REAL[5] / 10.0;
   #RAnalogArray[6] := #TYPE_800_AI_REAL[6] / 10.0;
   #RAnalogArray[7] := #TYPE_800_AI_REAL[7] / 10.0;
   #RAnalogArray[8] := #TYPE_800_AI_REAL[8] / 10.0;
   #RAnalogArray[9] := #TYPE_800_AI_REAL[9] / 10.0;
   #RAnalogArray[10] := #TYPE_800_AI_REAL[10] / 10.0;
   #RAnalogArray[11] := #TYPE_800_AI_REAL[11] / 10.0;
   #RAnalogArray[12] := #TYPE_800_AI_REAL[12] / 10.0;
   #RAnalogArray[13] := #TYPE_800_AI_REAL[13] / 10.0;
   #RAnalogArray[14] := #TYPE_800_AI_REAL[14] / 10.0;
   #RAnalogArray[15] := #TYPE_800_AI_REAL[15] / 10.0;
   #RAnalogArray[16] := #TYPE_800_AI_REAL[16] / 10.0;
   #RAnalogArray[17] := #TYPE_800_AI_REAL[17] / 10.0;
   #RAnalogArray[18] := #TYPE_800_AI_REAL[18] / 10.0;
   #RAnalogArray[19] := #TYPE_800_AI_REAL[19] / 10.0;
   #DummyBool := TRUE;
END_REGION

REGION Network 143
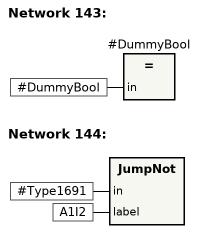
   A1I1:
   #DummyBool := #DummyBool;
END_REGION

REGION Network 144
   // no SCL statement known for JumpNot: written as a call
   JumpNot(in := #Type1691, label := A1I2);
END_REGION

REGION Network 145: Convert Analog to Floating Point
   // Transfer all Word data into Double Format and then to Real. Multiply with 10.0
   // SPC must be configured for sending processvalue with floating point 
   // representation.
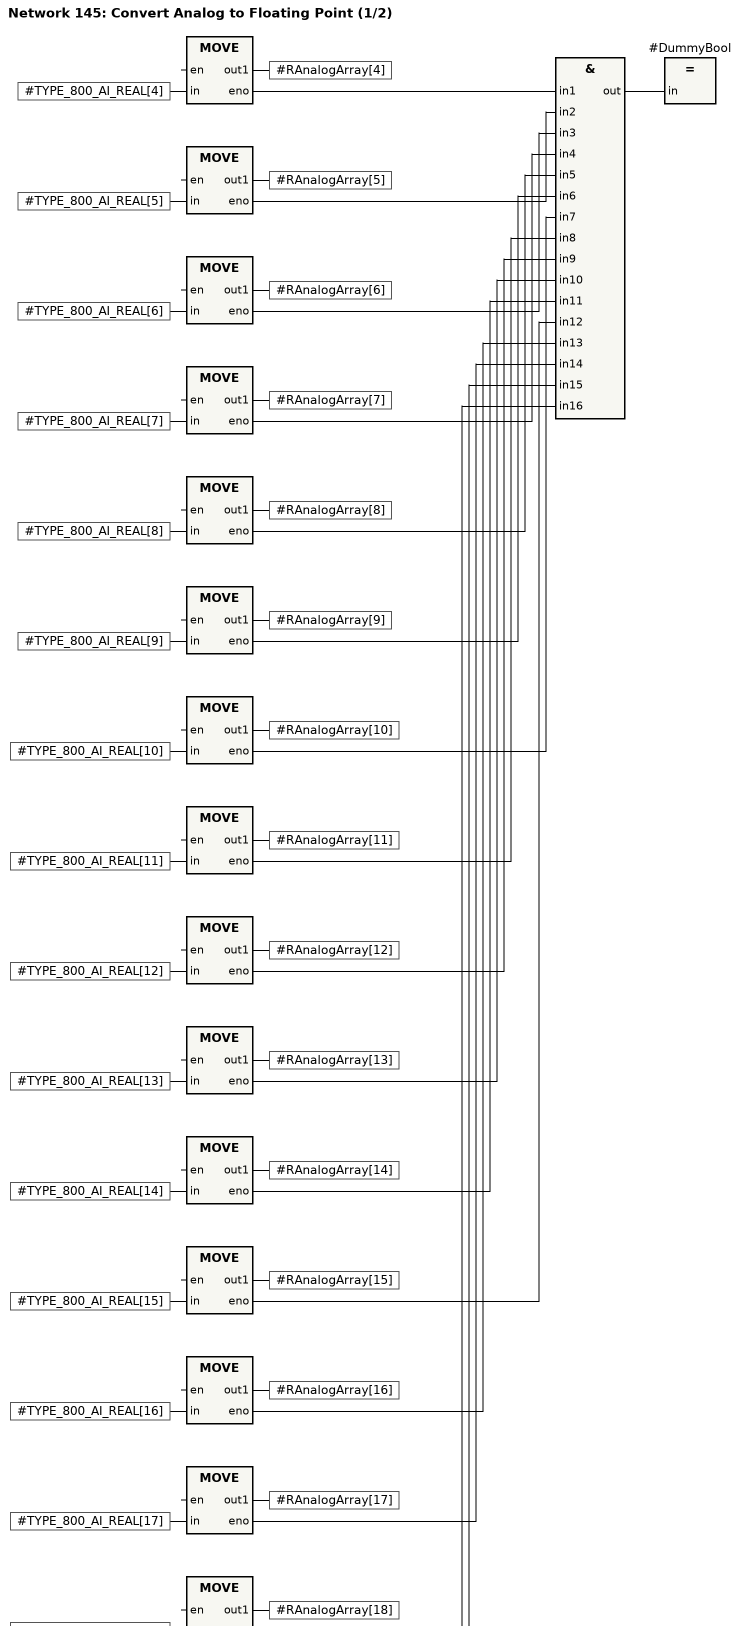
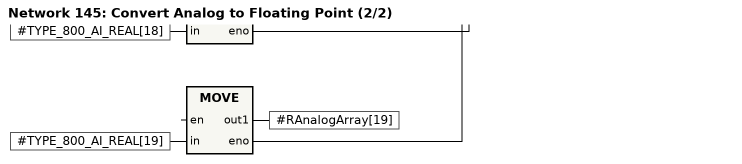
   #RAnalogArray[4] := #TYPE_800_AI_REAL[4];
   #RAnalogArray[5] := #TYPE_800_AI_REAL[5];
   #RAnalogArray[6] := #TYPE_800_AI_REAL[6];
   #RAnalogArray[7] := #TYPE_800_AI_REAL[7];
   #RAnalogArray[8] := #TYPE_800_AI_REAL[8];
   #RAnalogArray[9] := #TYPE_800_AI_REAL[9];
   #RAnalogArray[10] := #TYPE_800_AI_REAL[10];
   #RAnalogArray[11] := #TYPE_800_AI_REAL[11];
   #RAnalogArray[12] := #TYPE_800_AI_REAL[12];
   #RAnalogArray[13] := #TYPE_800_AI_REAL[13];
   #RAnalogArray[14] := #TYPE_800_AI_REAL[14];
   #RAnalogArray[15] := #TYPE_800_AI_REAL[15];
   #RAnalogArray[16] := #TYPE_800_AI_REAL[16];
   #RAnalogArray[17] := #TYPE_800_AI_REAL[17];
   #RAnalogArray[18] := #TYPE_800_AI_REAL[18];
   #RAnalogArray[19] := #TYPE_800_AI_REAL[19];
   #DummyBool := TRUE;
END_REGION

REGION Network 146
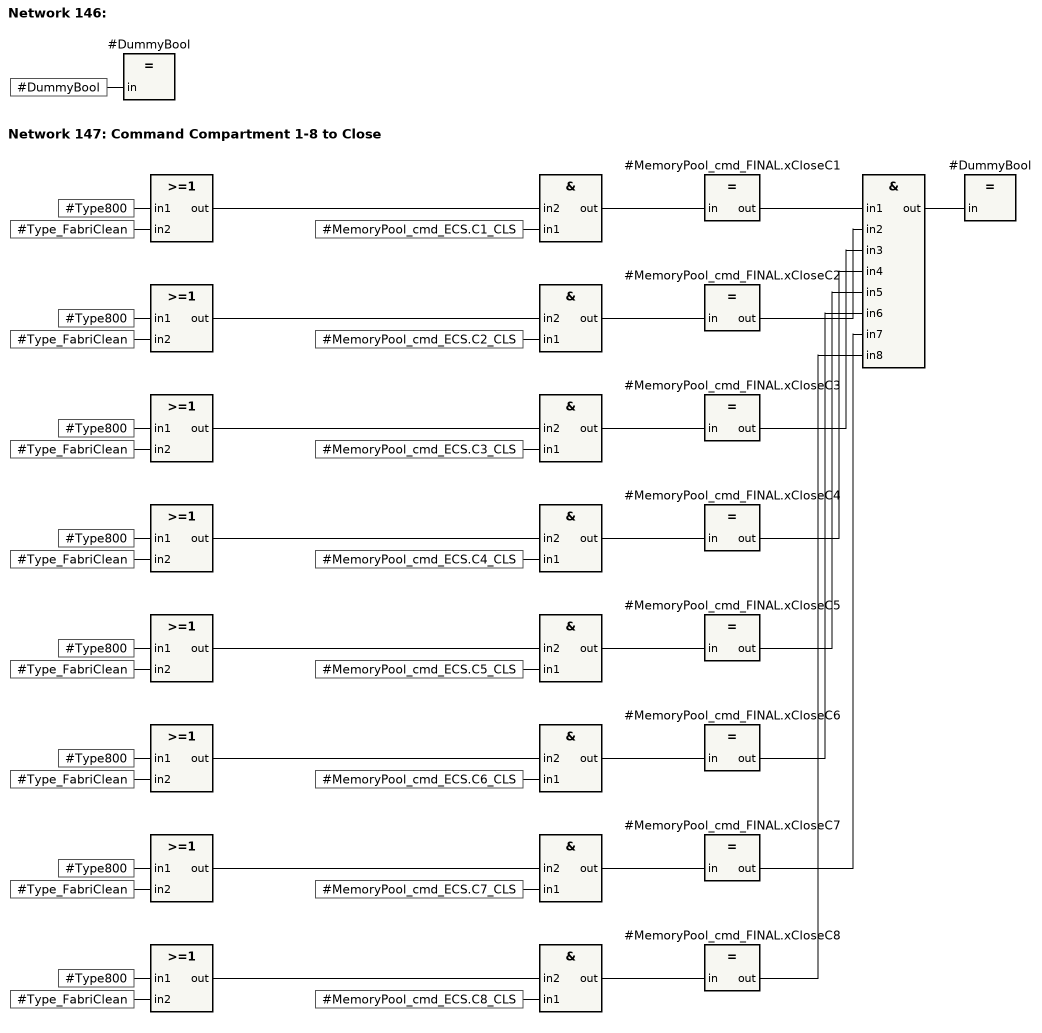
   A1I2:
   #DummyBool := #DummyBool;
END_REGION

REGION Network 147: Command Compartment 1-8 to Close
   #MemoryPool_cmd_FINAL.xCloseC1 := (#Type800 OR #Type_FabriClean) AND #MemoryPool_cmd_ECS.C1_CLS;
   #MemoryPool_cmd_FINAL.xCloseC2 := (#Type800 OR #Type_FabriClean) AND #MemoryPool_cmd_ECS.C2_CLS;
   #MemoryPool_cmd_FINAL.xCloseC3 := (#Type800 OR #Type_FabriClean) AND #MemoryPool_cmd_ECS.C3_CLS;
   #MemoryPool_cmd_FINAL.xCloseC4 := (#Type800 OR #Type_FabriClean) AND #MemoryPool_cmd_ECS.C4_CLS;
   #MemoryPool_cmd_FINAL.xCloseC5 := (#Type800 OR #Type_FabriClean) AND #MemoryPool_cmd_ECS.C5_CLS;
   #MemoryPool_cmd_FINAL.xCloseC6 := (#Type800 OR #Type_FabriClean) AND #MemoryPool_cmd_ECS.C6_CLS;
   #MemoryPool_cmd_FINAL.xCloseC7 := (#Type800 OR #Type_FabriClean) AND #MemoryPool_cmd_ECS.C7_CLS;
   #MemoryPool_cmd_FINAL.xCloseC8 := (#Type800 OR #Type_FabriClean) AND #MemoryPool_cmd_ECS.C8_CLS;
   #DummyBool := #MemoryPool_cmd_FINAL.xCloseC1 AND #MemoryPool_cmd_FINAL.xCloseC2 AND #MemoryPool_cmd_FINAL.xCloseC3 AND #MemoryPool_cmd_FINAL.xCloseC4 AND #MemoryPool_cmd_FINAL.xCloseC5 AND #MemoryPool_cmd_FINAL.xCloseC6 AND #MemoryPool_cmd_FINAL.xCloseC7 AND #MemoryPool_cmd_FINAL.xCloseC8;
END_REGION

REGION Network 148: Command Compartment 9-16 to Close
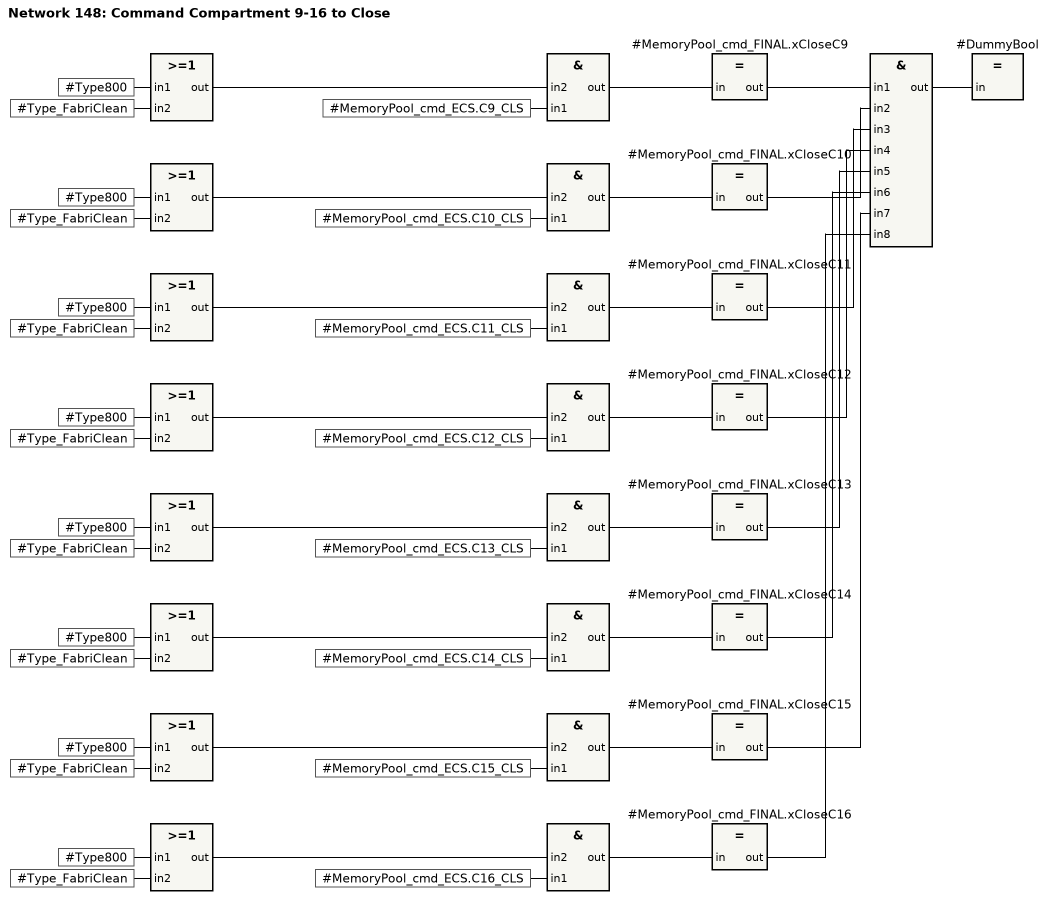
   #MemoryPool_cmd_FINAL.xCloseC9 := (#Type800 OR #Type_FabriClean) AND #MemoryPool_cmd_ECS.C9_CLS;
   #MemoryPool_cmd_FINAL.xCloseC10 := (#Type800 OR #Type_FabriClean) AND #MemoryPool_cmd_ECS.C10_CLS;
   #MemoryPool_cmd_FINAL.xCloseC11 := (#Type800 OR #Type_FabriClean) AND #MemoryPool_cmd_ECS.C11_CLS;
   #MemoryPool_cmd_FINAL.xCloseC12 := (#Type800 OR #Type_FabriClean) AND #MemoryPool_cmd_ECS.C12_CLS;
   #MemoryPool_cmd_FINAL.xCloseC13 := (#Type800 OR #Type_FabriClean) AND #MemoryPool_cmd_ECS.C13_CLS;
   #MemoryPool_cmd_FINAL.xCloseC14 := (#Type800 OR #Type_FabriClean) AND #MemoryPool_cmd_ECS.C14_CLS;
   #MemoryPool_cmd_FINAL.xCloseC15 := (#Type800 OR #Type_FabriClean) AND #MemoryPool_cmd_ECS.C15_CLS;
   #MemoryPool_cmd_FINAL.xCloseC16 := (#Type800 OR #Type_FabriClean) AND #MemoryPool_cmd_ECS.C16_CLS;
   #DummyBool := #MemoryPool_cmd_FINAL.xCloseC9 AND #MemoryPool_cmd_FINAL.xCloseC10 AND #MemoryPool_cmd_FINAL.xCloseC11 AND #MemoryPool_cmd_FINAL.xCloseC12 AND #MemoryPool_cmd_FINAL.xCloseC13 AND #MemoryPool_cmd_FINAL.xCloseC14 AND #MemoryPool_cmd_FINAL.xCloseC15 AND #MemoryPool_cmd_FINAL.xCloseC16;
END_REGION

REGION Network 149: Command Compartment 17-24 to Close
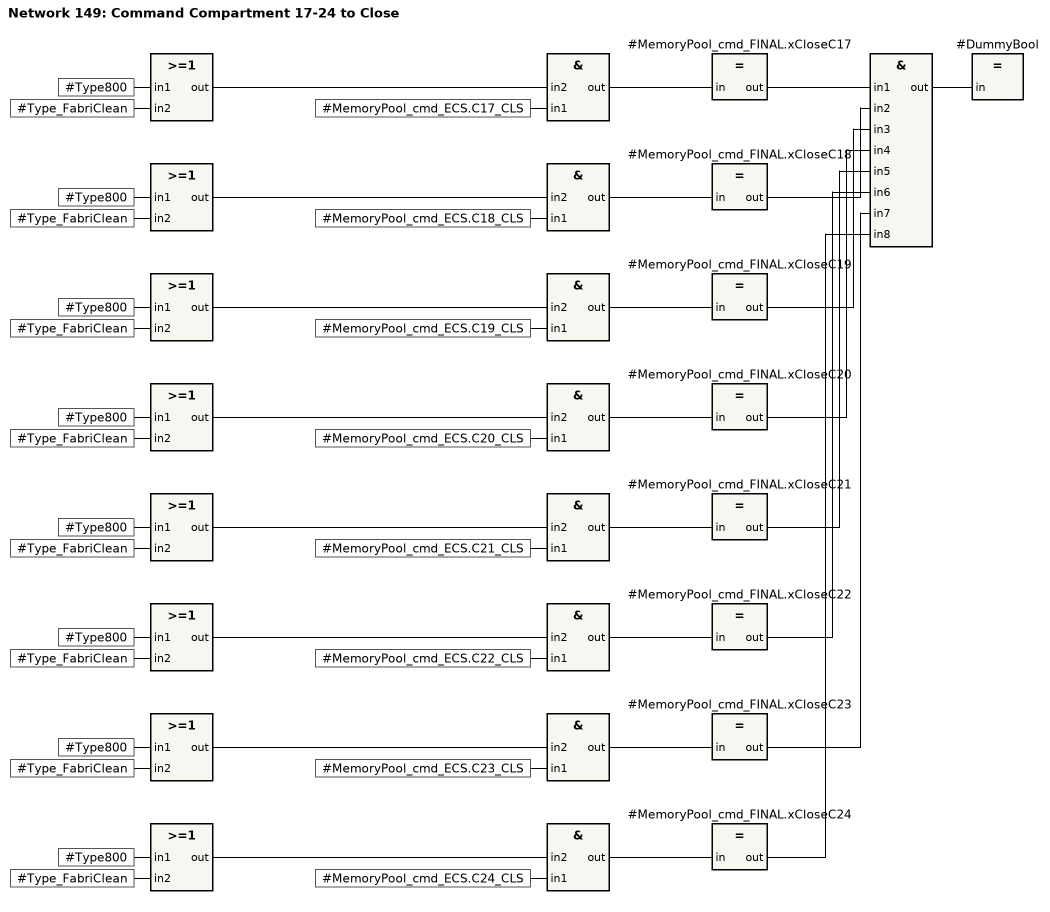
   #MemoryPool_cmd_FINAL.xCloseC17 := (#Type800 OR #Type_FabriClean) AND #MemoryPool_cmd_ECS.C17_CLS;
   #MemoryPool_cmd_FINAL.xCloseC18 := (#Type800 OR #Type_FabriClean) AND #MemoryPool_cmd_ECS.C18_CLS;
   #MemoryPool_cmd_FINAL.xCloseC19 := (#Type800 OR #Type_FabriClean) AND #MemoryPool_cmd_ECS.C19_CLS;
   #MemoryPool_cmd_FINAL.xCloseC20 := (#Type800 OR #Type_FabriClean) AND #MemoryPool_cmd_ECS.C20_CLS;
   #MemoryPool_cmd_FINAL.xCloseC21 := (#Type800 OR #Type_FabriClean) AND #MemoryPool_cmd_ECS.C21_CLS;
   #MemoryPool_cmd_FINAL.xCloseC22 := (#Type800 OR #Type_FabriClean) AND #MemoryPool_cmd_ECS.C22_CLS;
   #MemoryPool_cmd_FINAL.xCloseC23 := (#Type800 OR #Type_FabriClean) AND #MemoryPool_cmd_ECS.C23_CLS;
   #MemoryPool_cmd_FINAL.xCloseC24 := (#Type800 OR #Type_FabriClean) AND #MemoryPool_cmd_ECS.C24_CLS;
   #DummyBool := #MemoryPool_cmd_FINAL.xCloseC17 AND #MemoryPool_cmd_FINAL.xCloseC18 AND #MemoryPool_cmd_FINAL.xCloseC19 AND #MemoryPool_cmd_FINAL.xCloseC20 AND #MemoryPool_cmd_FINAL.xCloseC21 AND #MemoryPool_cmd_FINAL.xCloseC22 AND #MemoryPool_cmd_FINAL.xCloseC23 AND #MemoryPool_cmd_FINAL.xCloseC24;
END_REGION

REGION Network 150: Command Compartment 1-8 to Clean
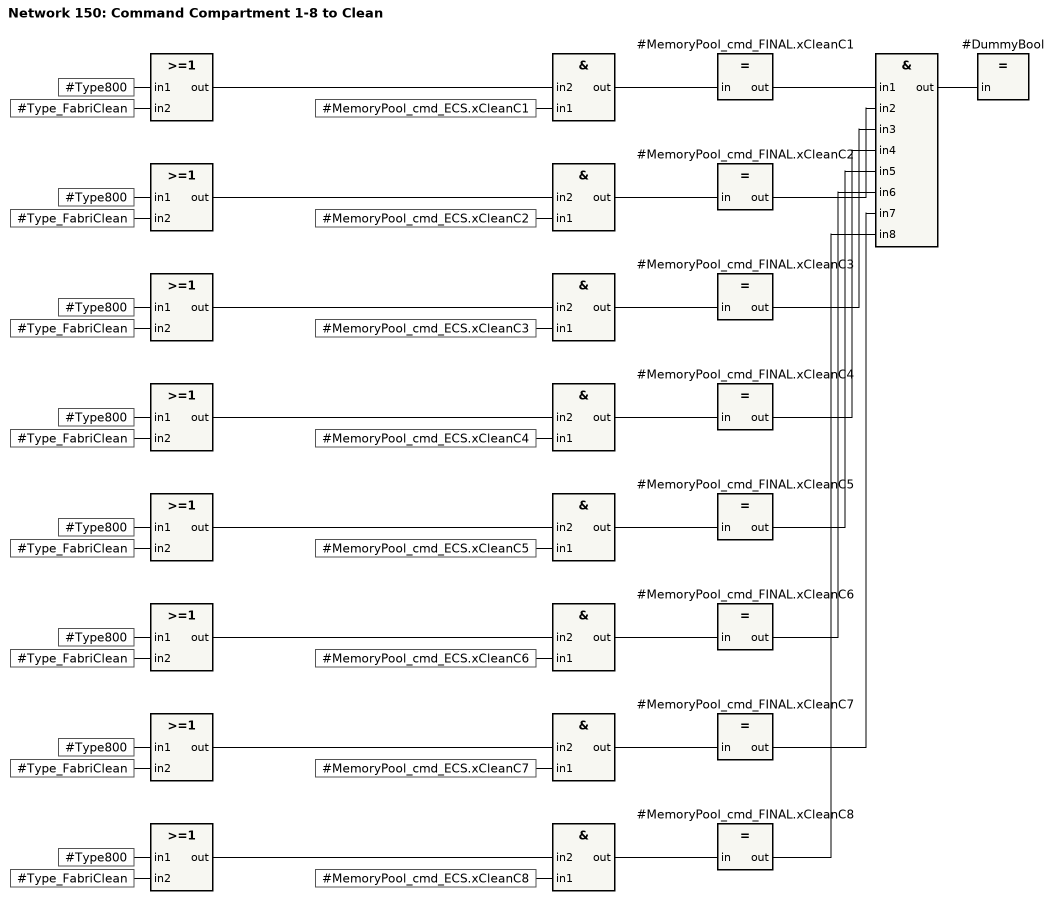
   #MemoryPool_cmd_FINAL.xCleanC1 := (#Type800 OR #Type_FabriClean) AND #MemoryPool_cmd_ECS.xCleanC1;
   #MemoryPool_cmd_FINAL.xCleanC2 := (#Type800 OR #Type_FabriClean) AND #MemoryPool_cmd_ECS.xCleanC2;
   #MemoryPool_cmd_FINAL.xCleanC3 := (#Type800 OR #Type_FabriClean) AND #MemoryPool_cmd_ECS.xCleanC3;
   #MemoryPool_cmd_FINAL.xCleanC4 := (#Type800 OR #Type_FabriClean) AND #MemoryPool_cmd_ECS.xCleanC4;
   #MemoryPool_cmd_FINAL.xCleanC5 := (#Type800 OR #Type_FabriClean) AND #MemoryPool_cmd_ECS.xCleanC5;
   #MemoryPool_cmd_FINAL.xCleanC6 := (#Type800 OR #Type_FabriClean) AND #MemoryPool_cmd_ECS.xCleanC6;
   #MemoryPool_cmd_FINAL.xCleanC7 := (#Type800 OR #Type_FabriClean) AND #MemoryPool_cmd_ECS.xCleanC7;
   #MemoryPool_cmd_FINAL.xCleanC8 := (#Type800 OR #Type_FabriClean) AND #MemoryPool_cmd_ECS.xCleanC8;
   #DummyBool := #MemoryPool_cmd_FINAL.xCleanC1 AND #MemoryPool_cmd_FINAL.xCleanC2 AND #MemoryPool_cmd_FINAL.xCleanC3 AND #MemoryPool_cmd_FINAL.xCleanC4 AND #MemoryPool_cmd_FINAL.xCleanC5 AND #MemoryPool_cmd_FINAL.xCleanC6 AND #MemoryPool_cmd_FINAL.xCleanC7 AND #MemoryPool_cmd_FINAL.xCleanC8;
END_REGION

REGION Network 151: Command Compartment 9-16 to Clean
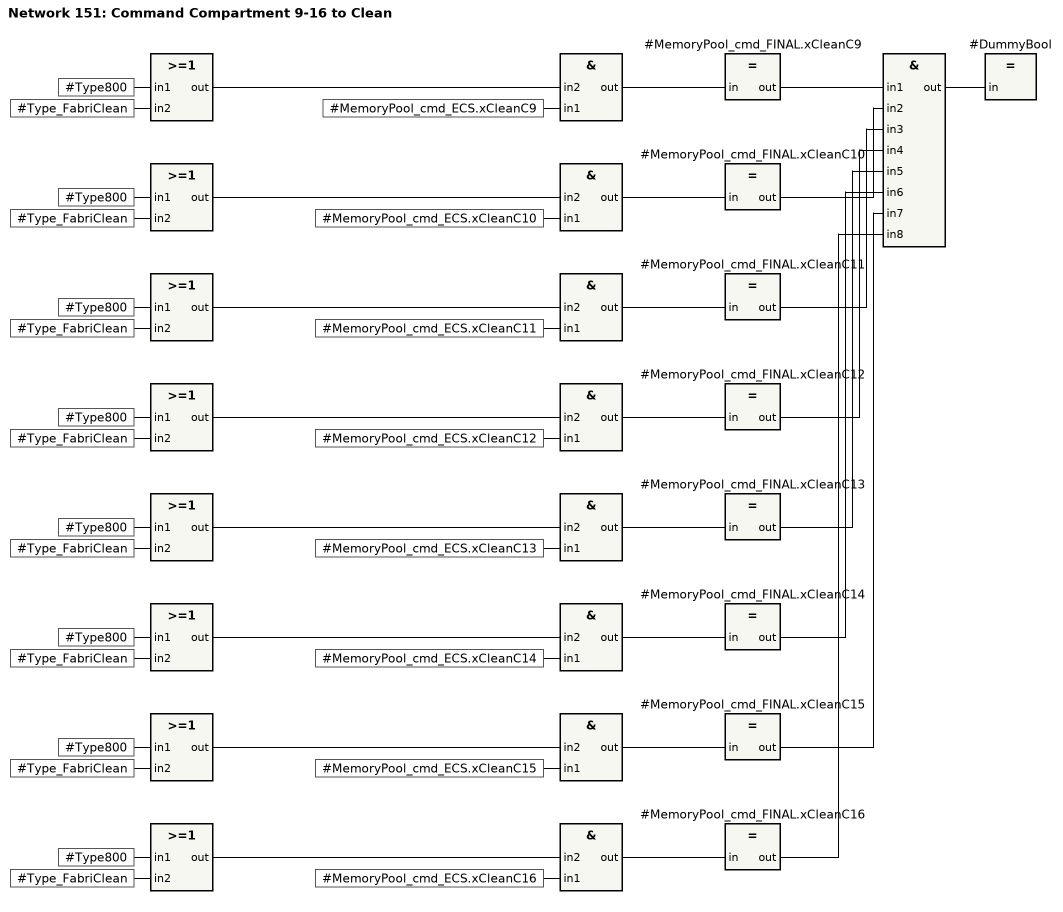
   #MemoryPool_cmd_FINAL.xCleanC9 := (#Type800 OR #Type_FabriClean) AND #MemoryPool_cmd_ECS.xCleanC9;
   #MemoryPool_cmd_FINAL.xCleanC10 := (#Type800 OR #Type_FabriClean) AND #MemoryPool_cmd_ECS.xCleanC10;
   #MemoryPool_cmd_FINAL.xCleanC11 := (#Type800 OR #Type_FabriClean) AND #MemoryPool_cmd_ECS.xCleanC11;
   #MemoryPool_cmd_FINAL.xCleanC12 := (#Type800 OR #Type_FabriClean) AND #MemoryPool_cmd_ECS.xCleanC12;
   #MemoryPool_cmd_FINAL.xCleanC13 := (#Type800 OR #Type_FabriClean) AND #MemoryPool_cmd_ECS.xCleanC13;
   #MemoryPool_cmd_FINAL.xCleanC14 := (#Type800 OR #Type_FabriClean) AND #MemoryPool_cmd_ECS.xCleanC14;
   #MemoryPool_cmd_FINAL.xCleanC15 := (#Type800 OR #Type_FabriClean) AND #MemoryPool_cmd_ECS.xCleanC15;
   #MemoryPool_cmd_FINAL.xCleanC16 := (#Type800 OR #Type_FabriClean) AND #MemoryPool_cmd_ECS.xCleanC16;
   #DummyBool := #MemoryPool_cmd_FINAL.xCleanC9 AND #MemoryPool_cmd_FINAL.xCleanC10 AND #MemoryPool_cmd_FINAL.xCleanC11 AND #MemoryPool_cmd_FINAL.xCleanC12 AND #MemoryPool_cmd_FINAL.xCleanC13 AND #MemoryPool_cmd_FINAL.xCleanC14 AND #MemoryPool_cmd_FINAL.xCleanC15 AND #MemoryPool_cmd_FINAL.xCleanC16;
END_REGION

REGION Network 152: Command Compartment 17-24 to Clean
